# B&R Automation Studio project MotionTestBenchMaster (part 46)

#### Itc_Filler.st
```iecst
ACTION FillerInput:
	(* Commands *)
	VAR_Machine.stFillerModule.iq_stCmd.i_xFillerAbsolutePositionSensor		:= MC_InputOutput.Network.Filler.Commands.FillerAbsolutePositionSensor; (*//V4.A.A.1.6.12e*)
	VAR_Machine.stFillerModule.iq_stCmd.i_xRinserFillerAbsolutePosSensor	:= MC_InputOutput.Network.Filler.Commands.RinserAbsolutePositionSensor; (*//V4.A.A.1.6.12e*)
	VAR_Machine.stFillerModule.iq_stCmd.i_xCapperAbsolutePositionSensor		:= MC_InputOutput.Network.Filler.Commands.CapperAbsolutePositionSensor; (*//V4.A.A.1.6.12e*)
	VAR_Machine.stFillerModule.iq_stCmd.i_xCrownerAbsolutePositionSensor	:= MC_InputOutput.Network.Filler.Commands.CrownerAbsolutePositionSensor; (*//V4.A.A.1.6.12e*)
	VAR_Machine.stFillerModule.iq_stCmd.i_xDoserAbsolutePositionSensor		:= MC_InputOutput.Network.Filler.Commands.DoserAbsolutePositionSensor; (*//V4.A.A.1.6.12e*)

	VAR_Machine.stFillerModule.iq_stCmd.i_xVelocityAxisStop				:= MC_InputOutput.Network.Filler.Commands.VelocityAxisStop;

	FOR uiAxisIndex := CST_FirstFillerModuleAxis TO CST_LastFillerModuleAxis DO
		VAR_Machine.stFillerModule.iq_astSubModuleAxis[uiAxisIndex].iq_stStatus.q_stMainAxisStatus.iq_xNotErrEncoder	:= MC_InputOutput.Safety.Filler.Commands.AxesDiag[uiAxisIndex].DI_NotErrENC;
		VAR_Machine.stFillerModule.iq_astSubModuleAxis[uiAxisIndex].iq_stStatus.q_stMainAxisStatus.iq_xOperational		:= MC_InputOutput.Safety.Filler.Commands.AxesDiag[uiAxisIndex].DI_Operational;
		(* Parameters *)
		IF uiAxisIndex >= 15 THEN
			VAR_Machine.stFillerModule.iq_astSubModuleAxis[uiAxisIndex].iq_stParam.i_rVelocityOffsetFactor		:= MC_InputOutput.Network.Filler.Parameters.OutletConveyorKs / 100.0;
		ELSE
			VAR_Machine.stFillerModule.iq_astSubModuleAxis[uiAxisIndex].iq_stParam.i_rVelocityOffsetFactor		:= MC_InputOutput.Network.Filler.Parameters.InletConveyorKs / 100.0;
		END_IF
	END_FOR

	VAR_Machine.stFillerModule.iq_stParameters.i_uiFillerAbsolutePositionOffset	:= MC_InputOutput.Network.Filler.Parameters.FillerAbsolutePositionOffset; (*//V4.A.A.1.6.12e*)
	VAR_Machine.stFillerModule.iq_stParameters.i_uiFillerStepsNumber			:= MC_InputOutput.Network.Filler.Parameters.FillerStepsNumber; (*//V4.A.A.1.6.12e*)
	VAR_Machine.stFillerModule.iq_stParameters.i_uiRinserAbsolutePositionOffset	:= MC_InputOutput.Network.Filler.Parameters.RinserAbsolutePositionOffset; (*//V4.A.A.1.6.12e*)
	VAR_Machine.stFillerModule.iq_stParameters.i_uiRinserStepsNumber			:= MC_InputOutput.Network.Filler.Parameters.RinserStepsNumber; (*//V4.A.A.1.6.12e*)
	VAR_Machine.stFillerModule.iq_stParameters.i_uiCapperAbsolutePositionOffset	:= MC_InputOutput.Network.Filler.Parameters.CapperAbsolutePositionOffset; (*//V4.A.A.1.6.12e*)
	VAR_Machine.stFillerModule.iq_stParameters.i_uiCapperStepsNumber			:= MC_InputOutput.Network.Filler.Parameters.CapperStepsNumber; (*//V4.A.A.1.6.12e*)
	VAR_Machine.stFillerModule.iq_stParameters.i_uiCrownerAbsolutePosOffset		:= MC_InputOutput.Network.Filler.Parameters.CrownerAbsolutePositionOffset; (*//V4.A.A.1.6.12e*)
	VAR_Machine.stFillerModule.iq_stParameters.i_uiCrownerStepsNumber			:= MC_InputOutput.Network.Filler.Parameters.CrownerStepsNumber; (*//V4.A.A.1.6.12e*)
	VAR_Machine.stFillerModule.iq_stParameters.i_uiDoserPositionOffset			:= MC_InputOutput.Network.Filler.Parameters.DoserAbsolutePositionOffset; (*//V4.A.A.1.6.12e*)
	VAR_Machine.stFillerModule.iq_stParameters.i_uiDoserStepsNumber				:= MC_InputOutput.Network.Filler.Parameters.DoserStepsNumber; (*//V4.A.A.1.6.12e*)

		(*Disable axis Rinser command*)
	VAR_Machine.stFillerModule.iq_astSubModuleAxis[CFG_MC.Mechanical.ReferenceId.Rinser].iq_stCmd.i_xDisableAxis	:= MC_InputOutput.Network.Filler.Commands.DisableRinserAxis;//V4.A.A.1.7.0
	(*Disable axis Doser command*)
	VAR_Machine.stFillerModule.iq_astSubModuleAxis[CFG_MC.Mechanical.ReferenceId.Doser].iq_stCmd.i_xDisableAxis		:= MC_InputOutput.Network.Filler.Commands.DisableDoserAxis;//v999 test
	(*Disable axis Filler command*)
	VAR_Machine.stFillerModule.iq_astSubModuleAxis[CFG_MC.Mechanical.ReferenceId.Filler].iq_stCmd.i_xDisableAxis		:= MC_InputOutput.Network.Filler.Commands.DisableFillerAxis;//v999 test

//	VAR_Machine.stFillerModule.iq_astSubModuleAxis[CST_Inlet10].iq_stCmd.i_xDisableAxis := MC_InputOutput.Network.Filler.Commands.MotorDisableIndex[CST_Inlet10] AND VAR_Machine.stFillerModule.iq_astSubModuleAxis[CST_Inlet10].iq_stStatus.q_stMainAxisStatus.q_xAxisReal;
//	VAR_Machine.stFillerModule.iq_astSubModuleAxis[CST_Inlet09].iq_stCmd.i_xDisableAxis := MC_InputOutput.Network.Filler.Commands.MotorDisableIndex[CST_Inlet09] AND VAR_Machine.stFillerModule.iq_astSubModuleAxis[CST_Inlet09].iq_stStatus.q_stMainAxisStatus.q_xAxisReal;
//	VAR_Machine.stFillerModule.iq_astSubModuleAxis[CST_Inlet08].iq_stCmd.i_xDisableAxis := MC_InputOutput.Network.Filler.Commands.MotorDisableIndex[CST_Inlet08] AND VAR_Machine.stFillerModule.iq_astSubModuleAxis[CST_Inlet08].iq_stStatus.q_stMainAxisStatus.q_xAxisReal;
//	VAR_Machine.stFillerModule.iq_astSubModuleAxis[CST_Inlet07].iq_stCmd.i_xDisableAxis := MC_InputOutput.Network.Filler.Commands.MotorDisableIndex[CST_Inlet07] AND VAR_Machine.stFillerModule.iq_astSubModuleAxis[CST_Inlet07].iq_stStatus.q_stMainAxisStatus.q_xAxisReal;
//	VAR_Machine.stFillerModule.iq_astSubModuleAxis[CST_Inlet06].iq_stCmd.i_xDisableAxis := MC_InputOutput.Network.Filler.Commands.MotorDisableIndex[CST_Inlet06] AND VAR_Machine.stFillerModule.iq_astSubModuleAxis[CST_Inlet06].iq_stStatus.q_stMainAxisStatus.q_xAxisReal;
//	VAR_Machine.stFillerModule.iq_astSubModuleAxis[CST_Inlet05].iq_stCmd.i_xDisableAxis := MC_InputOutput.Network.Filler.Commands.MotorDisableIndex[CST_Inlet05] AND VAR_Machine.stFillerModule.iq_astSubModuleAxis[CST_Inlet05].iq_stStatus.q_stMainAxisStatus.q_xAxisReal;
//	VAR_Machine.stFillerModule.iq_astSubModuleAxis[CST_Inlet04].iq_stCmd.i_xDisableAxis := MC_InputOutput.Network.Filler.Commands.MotorDisableIndex[CST_Inlet04] AND VAR_Machine.stFillerModule.iq_astSubModuleAxis[CST_Inlet04].iq_stStatus.q_stMainAxisStatus.q_xAxisReal;
//	VAR_Machine.stFillerModule.iq_astSubModuleAxis[CST_Inlet03].iq_stCmd.i_xDisableAxis := MC_InputOutput.Network.Filler.Commands.MotorDisableIndex[CST_Inlet03] AND VAR_Machine.stFillerModule.iq_astSubModuleAxis[CST_Inlet03].iq_stStatus.q_stMainAxisStatus.q_xAxisReal;
//	VAR_Machine.stFillerModule.iq_astSubModuleAxis[CST_Inlet02].iq_stCmd.i_xDisableAxis := MC_InputOutput.Network.Filler.Commands.MotorDisableIndex[CST_Inlet02] AND VAR_Machine.stFillerModule.iq_astSubModuleAxis[CST_Inlet02].iq_stStatus.q_stMainAxisStatus.q_xAxisReal;
//	VAR_Machine.stFillerModule.iq_astSubModuleAxis[CST_Inlet01].iq_stCmd.i_xDisableAxis := MC_InputOutput.Network.Filler.Commands.MotorDisableIndex[CST_Inlet01] AND VAR_Machine.stFillerModule.iq_astSubModuleAxis[CST_Inlet01].iq_stStatus.q_stMainAxisStatus.q_xAxisReal;
//	VAR_Machine.stFillerModule.iq_astSubModuleAxis[CST_MainAxis].iq_stCmd.i_xDisableAxis := MC_InputOutput.Network.Filler.Commands.MotorDisableIndex[CST_MainAxis] AND VAR_Machine.stFillerModule.iq_astSubModuleAxis[CST_MainAxis].iq_stStatus.q_stMainAxisStatus.q_xAxisReal;
//	VAR_Machine.stFillerModule.iq_astSubModuleAxis[CST_Outlet01].iq_stCmd.i_xDisableAxis := MC_InputOutput.Network.Filler.Commands.MotorDisableIndex[CST_Outlet01] AND VAR_Machine.stFillerModule.iq_astSubModuleAxis[CST_Outlet01].iq_stStatus.q_stMainAxisStatus.q_xAxisReal;
//	VAR_Machine.stFillerModule.iq_astSubModuleAxis[CST_Outlet02].iq_stCmd.i_xDisableAxis := MC_InputOutput.Network.Filler.Commands.MotorDisableIndex[CST_Outlet02] AND VAR_Machine.stFillerModule.iq_astSubModuleAxis[CST_Outlet02].iq_stStatus.q_stMainAxisStatus.q_xAxisReal;
//	VAR_Machine.stFillerModule.iq_astSubModuleAxis[CST_Outlet03].iq_stCmd.i_xDisableAxis := MC_InputOutput.Network.Filler.Commands.MotorDisableIndex[CST_Outlet03] AND VAR_Machine.stFillerModule.iq_astSubModuleAxis[CST_Outlet03].iq_stStatus.q_stMainAxisStatus.q_xAxisReal;
//	VAR_Machine.stFillerModule.iq_astSubModuleAxis[CST_Outlet04].iq_stCmd.i_xDisableAxis := MC_InputOutput.Network.Filler.Commands.MotorDisableIndex[CST_Outlet04] AND VAR_Machine.stFillerModule.iq_astSubModuleAxis[CST_Outlet04].iq_stStatus.q_stMainAxisStatus.q_xAxisReal;
//	VAR_Machine.stFillerModule.iq_astSubModuleAxis[CST_Outlet05].iq_stCmd.i_xDisableAxis := MC_InputOutput.Network.Filler.Commands.MotorDisableIndex[CST_Outlet05] AND VAR_Machine.stFillerModule.iq_astSubModuleAxis[CST_Outlet05].iq_stStatus.q_stMainAxisStatus.q_xAxisReal;
//	VAR_Machine.stFillerModule.iq_astSubModuleAxis[CST_Outlet06].iq_stCmd.i_xDisableAxis := MC_InputOutput.Network.Filler.Commands.MotorDisableIndex[CST_Outlet06] AND VAR_Machine.stFillerModule.iq_astSubModuleAxis[CST_Outlet06].iq_stStatus.q_stMainAxisStatus.q_xAxisReal;

	VAR_Machine.stFillerModule.iq_astSubModuleAxis[CST_MainAxis].iq_stParam.i_rTorqueErrorThreshold	:= MC_InputOutput.Network.Filler.Parameters.TorqueError.Main;
	FOR uiAxisIndex := 1 TO 10 DO
		VAR_Machine.stFillerModule.iq_astSubModuleAxis[(uiAxisIndex - 1) +  CST_FirstFillerModuleAxis].iq_stParam.i_rTorqueErrorThreshold	:= MC_InputOutput.Network.Filler.Parameters.TorqueError.In[uiAxisIndex];
	END_FOR

	FOR uiAxisIndex := 1 TO 6 DO
		VAR_Machine.stFillerModule.iq_astSubModuleAxis[(uiAxisIndex) + CST_MainAxis].iq_stParam.i_rTorqueErrorThreshold	:= MC_InputOutput.Network.Filler.Parameters.TorqueError.Out[uiAxisIndex];
	END_FOR
END_ACTION

ACTION FillerOutput:
	(* Filler status *)
	MC_InputOutput.Network.Filler.Status.Velocity						:= VAR_Machine.stFillerModule.iq_stStatus.q_rVelocity * 10.0;
	MC_InputOutput.Network.Filler.Status.FillerAbsolutePosition			:= VAR_Machine.stFillerModule.iq_stStatus.q_lrFillerAbsolutePosition; (*//V4.A.A.1.6.12e*)
	MC_InputOutput.Network.Filler.Status.RinserAbsolutePosition			:= VAR_Machine.stFillerModule.iq_stStatus.q_lrRinserAbsolutePosition; (*//V4.A.A.1.6.12e*)
	MC_InputOutput.Network.Filler.Status.CapperAbsolutePosition			:= VAR_Machine.stFillerModule.iq_stStatus.q_lrCapperAbsolutePosition; (*//V4.A.A.1.6.12e*)
	MC_InputOutput.Network.Filler.Status.CrownerAbsolutePosition		:= VAR_Machine.stFillerModule.iq_stStatus.q_lrCrownerAbsolutePosition; (*//V4.A.A.1.6.12e*)
	MC_InputOutput.Network.Filler.Status.DoserAbsolutePosition			:= VAR_Machine.stFillerModule.iq_stStatus.q_lrDoserAbsolutePosition; (*//V4.A.A.1.6.12e*)

	MC_InputOutput.Network.Filler.Status.ModuleHomed					:= VAR_Machine.stFillerModule.iq_stStatus.q_xModuleHomed;
	MC_InputOutput.Network.Filler.Status.ModuleInPosition;
	MC_InputOutput.Network.Filler.Status.ModulePowered					:= VAR_Machine.stFillerModule.iq_stStatus.q_xModulePowered;
	MC_InputOutput.Network.Filler.Status.ModuleReal						:= VAR_Machine.stFillerModule.iq_stStatus.q_xModuleReal;
	MC_InputOutput.Network.Filler.Status.ModuleRunning					:= SEL(VAR_Machine.iq_stStatus.q_xMultiModalityActive, VAR_Machine.iq_stStatus.q_xMachineStartFbk, VAR_Machine.stFillerModule.iq_stStatus.q_xModuleStartFbk);
	MC_InputOutput.Network.Filler.Status.ModuleNotInitialized			:= NOT VAR_Machine.stFillerModule.iq_stStatus.q_xInitDone;

	MC_InputOutput.Network.Filler.Status.AutoActive						:= VAR_Machine.stFillerModule.iq_stStatus.q_xAutoMultiActive;
	MC_InputOutput.Network.Filler.Status.ModuleJogActive				:= VAR_Machine.stFillerModule.iq_stStatus.q_xJogMultiActive;
	MC_InputOutput.Network.Filler.Status.SlowMotionActive				:= VAR_Machine.stFillerModule.iq_stStatus.q_xSlowMotionActive;

	MC_InputOutput.Network.Filler.Status.AutoCmdFeedback				:= VAR_Machine.stFillerModule.iq_stStatus.q_xAutoMultiActive AND VAR_Machine.stFillerModule.iq_stCmd.i_xStart;
	MC_InputOutput.Network.Filler.Status.JogCmdFeedback					:= VAR_Machine.stFillerModule.iq_stStatus.q_xJogMultiActive AND VAR_Machine.stFillerModule.iq_stCmd.i_xJogPB;

	MC_InputOutput.Network.Filler.Status.CarouselReal				:= VAR_Machine.stFillerModule.iq_astSubModuleAxis[CST_MainAxis].iq_stStatus.q_stMainAxisStatus.q_xAxisReal;
	MC_InputOutput.Network.Filler.Status.In01Real					:= VAR_Machine.stFillerModule.iq_astSubModuleAxis[CST_Inlet01].iq_stStatus.q_stMainAxisStatus.q_xAxisReal;
	MC_InputOutput.Network.Filler.Status.In02Real					:= VAR_Machine.stFillerModule.iq_astSubModuleAxis[CST_Inlet02].iq_stStatus.q_stMainAxisStatus.q_xAxisReal;
	MC_InputOutput.Network.Filler.Status.In03Real					:= VAR_Machine.stFillerModule.iq_astSubModuleAxis[CST_Inlet03].iq_stStatus.q_stMainAxisStatus.q_xAxisReal;
	MC_InputOutput.Network.Filler.Status.In04Real					:= VAR_Machine.stFillerModule.iq_astSubModuleAxis[CST_Inlet04].iq_stStatus.q_stMainAxisStatus.q_xAxisReal;
	MC_InputOutput.Network.Filler.Status.In05Real					:= VAR_Machine.stFillerModule.iq_astSubModuleAxis[CST_Inlet05].iq_stStatus.q_stMainAxisStatus.q_xAxisReal;
	MC_InputOutput.Network.Filler.Status.In06Real					:= VAR_Machine.stFillerModule.iq_astSubModuleAxis[CST_Inlet06].iq_stStatus.q_stMainAxisStatus.q_xAxisReal;
	MC_InputOutput.Network.Filler.Status.In07Real					:= VAR_Machine.stFillerModule.iq_astSubModuleAxis[CST_Inlet07].iq_stStatus.q_stMainAxisStatus.q_xAxisReal;
	MC_InputOutput.Network.Filler.Status.In08Real					:= VAR_Machine.stFillerModule.iq_astSubModuleAxis[CST_Inlet08].iq_stStatus.q_stMainAxisStatus.q_xAxisReal;
	MC_InputOutput.Network.Filler.Status.In09Real					:= VAR_Machine.stFillerModule.iq_astSubModuleAxis[CST_Inlet09].iq_stStatus.q_stMainAxisStatus.q_xAxisReal;
	MC_InputOutput.Network.Filler.Status.In10Real					:= VAR_Machine.stFillerModule.iq_astSubModuleAxis[CST_Inlet10].iq_stStatus.q_stMainAxisStatus.q_xAxisReal;
	MC_InputOutput.Network.Filler.Status.Out01Real					:= VAR_Machine.stFillerModule.iq_astSubModuleAxis[CST_Outlet01].iq_stStatus.q_stMainAxisStatus.q_xAxisReal;
	MC_InputOutput.Network.Filler.Status.Out02Real					:= VAR_Machine.stFillerModule.iq_astSubModuleAxis[CST_Outlet02].iq_stStatus.q_stMainAxisStatus.q_xAxisReal;
	MC_InputOutput.Network.Filler.Status.Out03Real					:= VAR_Machine.stFillerModule.iq_astSubModuleAxis[CST_Outlet03].iq_stStatus.q_stMainAxisStatus.q_xAxisReal;
	MC_InputOutput.Network.Filler.Status.Out04Real					:= VAR_Machine.stFillerModule.iq_astSubModuleAxis[CST_Outlet04].iq_stStatus.q_stMainAxisStatus.q_xAxisReal;
	MC_InputOutput.Network.Filler.Status.Out05Real					:= VAR_Machine.stFillerModule.iq_astSubModuleAxis[CST_Outlet05].iq_stStatus.q_stMainAxisStatus.q_xAxisReal;
	MC_InputOutput.Network.Filler.Status.Out06Real					:= VAR_Machine.stFillerModule.iq_astSubModuleAxis[CST_Outlet06].iq_stStatus.q_stMainAxisStatus.q_xAxisReal;

	MC_InputOutput.Network.Filler.Status.FillerAbsolutePositionValid			:= VAR_Machine.stFillerModule.iq_stStatus.q_xFillerAbsolutePositionValid; (*//V4.A.A.1.6.12e*)
	MC_InputOutput.Network.Filler.Status.RinserAbsolutePositionValid			:= VAR_Machine.stFillerModule.iq_stStatus.q_xRinserAbsolutePositionValid; (*//V4.A.A.1.6.12e*)
	MC_InputOutput.Network.Filler.Status.CapperAbsolutePositionValid			:= VAR_Machine.stFillerModule.iq_stStatus.q_xCapperAbsolutePositionValid; (*//V4.A.A.1.6.12e*)
	MC_InputOutput.Network.Filler.Status.CrownerAbsolutePositionValid			:= VAR_Machine.stFillerModule.iq_stStatus.q_xCrownerAbsolutePositionValid; (*//V4.A.A.1.6.12e*)
	MC_InputOutput.Network.Filler.Status.DoserAbsolutePositionValid				:= VAR_Machine.stFillerModule.iq_stStatus.q_xDoserAbsolutePositionValid; (*//V4.A.A.1.6.12e*)

	(* Disable Motor Filler Module Status ----------------------------*)

		(* Disabel Axis FeedBack *) //V4.A.A.1.7.0 Motion
	MC_InputOutput.Network.Filler.Status.DoserAxisDisabled						:= VAR_Machine.stFillerModule.iq_astSubModuleAxis[CFG_MC.Mechanical.ReferenceId.Doser].iq_stStatus.q_stMainAxisStatus.q_xAxisDisabled;
	MC_InputOutput.Network.Filler.Status.RinserAxisDisabled						:= VAR_Machine.stFillerModule.iq_astSubModuleAxis[CFG_MC.Mechanical.ReferenceId.Rinser].iq_stStatus.q_stMainAxisStatus.q_xAxisDisabled;

//	MC_InputOutput.Network.Filler.Status.AxisDisabledFeedBack[CST_Inlet10]		:= VAR_Machine.stFillerModule.iq_astSubModuleAxis[CST_Inlet10].iq_stStatus.q_stMainAxisStatus.q_xAxisDisabled;
//	MC_InputOutput.Network.Filler.Status.AxisDisabledFeedBack[CST_Inlet09]		:= VAR_Machine.stFillerModule.iq_astSubModuleAxis[CST_Inlet09].iq_stStatus.q_stMainAxisStatus.q_xAxisDisabled;
//	MC_InputOutput.Network.Filler.Status.AxisDisabledFeedBack[CST_Inlet08]		:= VAR_Machine.stFillerModule.iq_astSubModuleAxis[CST_Inlet08].iq_stStatus.q_stMainAxisStatus.q_xAxisDisabled;
//	MC_InputOutput.Network.Filler.Status.AxisDisabledFeedBack[CST_Inlet07]		:= VAR_Machine.stFillerModule.iq_astSubModuleAxis[CST_Inlet07].iq_stStatus.q_stMainAxisStatus.q_xAxisDisabled;
//	MC_InputOutput.Network.Filler.Status.AxisDisabledFeedBack[CST_Inlet06]		:= VAR_Machine.stFillerModule.iq_astSubModuleAxis[CST_Inlet06].iq_stStatus.q_stMainAxisStatus.q_xAxisDisabled;
//	MC_InputOutput.Network.Filler.Status.AxisDisabledFeedBack[CST_Inlet05]		:= VAR_Machine.stFillerModule.iq_astSubModuleAxis[CST_Inlet05].iq_stStatus.q_stMainAxisStatus.q_xAxisDisabled;
//	MC_InputOutput.Network.Filler.Status.AxisDisabledFeedBack[CST_Inlet04]		:= VAR_Machine.stFillerModule.iq_astSubModuleAxis[CST_Inlet04].iq_stStatus.q_stMainAxisStatus.q_xAxisDisabled;
//	MC_InputOutput.Network.Filler.Status.AxisDisabledFeedBack[CST_Inlet03]		:= VAR_Machine.stFillerModule.iq_astSubModuleAxis[CST_Inlet03].iq_stStatus.q_stMainAxisStatus.q_xAxisDisabled;
//	MC_InputOutput.Network.Filler.Status.AxisDisabledFeedBack[CST_Inlet02]		:= VAR_Machine.stFillerModule.iq_astSubModuleAxis[CST_Inlet02].iq_stStatus.q_stMainAxisStatus.q_xAxisDisabled;
//	MC_InputOutput.Network.Filler.Status.AxisDisabledFeedBack[CST_Inlet01]		:= VAR_Machine.stFillerModule.iq_astSubModuleAxis[CST_Inlet01].iq_stStatus.q_stMainAxisStatus.q_xAxisDisabled;
//	MC_InputOutput.Network.Filler.Status.AxisDisabledFeedBack[CST_MainAxis]		:= VAR_Machine.stFillerModule.iq_astSubModuleAxis[CST_MainAxis].iq_stStatus.q_stMainAxisStatus.q_xAxisDisabled;
//	MC_InputOutput.Network.Filler.Status.AxisDisabledFeedBack[CST_Outlet01]		:= VAR_Machine.stFillerModule.iq_astSubModuleAxis[CST_Outlet01].iq_stStatus.q_stMainAxisStatus.q_xAxisDisabled;
//	MC_InputOutput.Network.Filler.Status.AxisDisabledFeedBack[CST_Outlet02]		:= VAR_Machine.stFillerModule.iq_astSubModuleAxis[CST_Outlet02].iq_stStatus.q_stMainAxisStatus.q_xAxisDisabled;
//	MC_InputOutput.Network.Filler.Status.AxisDisabledFeedBack[CST_Outlet03]		:= VAR_Machine.stFillerModule.iq_astSubModuleAxis[CST_Outlet03].iq_stStatus.q_stMainAxisStatus.q_xAxisDisabled;
//	MC_InputOutput.Network.Filler.Status.AxisDisabledFeedBack[CST_Outlet04]		:= VAR_Machine.stFillerModule.iq_astSubModuleAxis[CST_Outlet04].iq_stStatus.q_stMainAxisStatus.q_xAxisDisabled;
//	MC_InputOutput.Network.Filler.Status.AxisDisabledFeedBack[CST_Outlet05]		:= VAR_Machine.stFillerModule.iq_astSubModuleAxis[CST_Outlet05].iq_stStatus.q_stMainAxisStatus.q_xAxisDisabled;
//	MC_InputOutput.Network.Filler.Status.AxisDisabledFeedBack[CST_Outlet06]		:= VAR_Machine.stFillerModule.iq_astSubModuleAxis[CST_Outlet06].iq_stStatus.q_stMainAxisStatus.q_xAxisDisabled;

	(* Button Enable *)
	MC_InputOutput.Network.Filler.Status.EnableAutoModality				:= NOT VAR_Machine.stFillerModule.iq_stStatus.q_xReactionActive;
	MC_InputOutput.Network.Filler.Status.EnableJogModality				:= VAR_Machine.stFillerModule.iq_stStatus.q_xModuleStopped AND
																			NOT VAR_Machine.stFillerModule.iq_stStatus.q_xReactionActive;

	(* Exception *)
	(* Main axis exception *)
	MC_InputOutput.Network.Filler.Exceptions.CarouselNotInOpException			:= NOT VAR_Machine.stFillerModule.iq_astSubModuleAxis[CST_MainAxis].iq_stStatus.q_stMainAxisStatus.iq_xOperational;
	MC_InputOutput.Network.Filler.Exceptions.CarouselSafetyException			:= NOT MC_InputOutput.Safety.Filler.Commands.AxesDiag[CST_MainAxis].DI_NotErrFUNC;
	MC_InputOutput.Network.Filler.Exceptions.CarouselTorqueException			:= VAR_Machine.stFillerModule.iq_astSubModuleAxis[CST_MainAxis].iq_stStatus.q_stMainAxisStatus.q_xTorqueError;
	MC_InputOutput.Network.Filler.Exceptions.CarouselTrackException				:= VAR_Machine.stFillerModule.iq_astSubModuleAxis[CST_MainAxis].iq_stStatus.q_stMainAxisStatus.q_xLagError;
	MC_InputOutput.Network.Filler.Exceptions.CarouselDriveException				:= VAR_Machine.stFillerModule.iq_astSubModuleAxis[CST_MainAxis].iq_stStatus.q_stMainAxisStatus.q_xError;
	MC_InputOutput.Network.Filler.Exceptions.CarouselHomeException				:= NOT VAR_Machine.stFillerModule.iq_astSubModuleAxis[CST_MainAxis].iq_stStatus.q_stMainAxisStatus.q_xIsHomed AND
																					VAR_Machine.stFillerModule.iq_astSubModuleAxis[CST_MainAxis].iq_stStatus.q_stMainAxisStatus.q_xInitDone;

	(* Inlet axis exception *)
	IF VAR_Machine.stFillerModule.iq_astSubModuleAxis[CST_Inlet01].iq_stStatus.q_stMainAxisStatus.q_xAxisReal THEN
		IF NOT CFG_MC.Axes.Filler.In[1].VelocityControl THEN
			MC_InputOutput.Network.Filler.Exceptions.Inlet01NotInOpException			:= NOT VAR_Machine.stFillerModule.iq_astSubModuleAxis[CST_Inlet01].iq_stStatus.q_stMainAxisStatus.iq_xOperational;
			MC_InputOutput.Network.Filler.Exceptions.Inlet01SafetyException				:= NOT MC_InputOutput.Safety.Filler.Commands.AxesDiag[CST_Inlet01].DI_NotErrFUNC;
		END_IF
		MC_InputOutput.Network.Filler.Exceptions.Inlet01TorqueException				:= VAR_Machine.stFillerModule.iq_astSubModuleAxis[CST_Inlet01].iq_stStatus.q_stMainAxisStatus.q_xTorqueError;
		MC_InputOutput.Network.Filler.Exceptions.Inlet01TrackException				:= VAR_Machine.stFillerModule.iq_astSubModuleAxis[CST_Inlet01].iq_stStatus.q_stMainAxisStatus.q_xLagError;
		MC_InputOutput.Network.Filler.Exceptions.Inlet01DriveException				:= VAR_Machine.stFillerModule.iq_astSubModuleAxis[CST_Inlet01].iq_stStatus.q_stMainAxisStatus.q_xError;
		MC_InputOutput.Network.Filler.Exceptions.Inlet01HomeException				:= NOT VAR_Machine.stFillerModule.iq_astSubModuleAxis[CST_Inlet01].iq_stStatus.q_stMainAxisStatus.q_xIsHomed AND
																						VAR_Machine.stFillerModule.iq_astSubModuleAxis[CST_Inlet01].iq_stStatus.q_stMainAxisStatus.q_xInitDone;
	END_IF

	IF VAR_Machine.stFillerModule.iq_astSubModuleAxis[CST_Inlet02].iq_stStatus.q_stMainAxisStatus.q_xAxisReal THEN
		IF NOT CFG_MC.Axes.Filler.In[2].VelocityControl THEN
			MC_InputOutput.Network.Filler.Exceptions.Inlet02NotInOpException			:= NOT VAR_Machine.stFillerModule.iq_astSubModuleAxis[CST_Inlet02].iq_stStatus.q_stMainAxisStatus.iq_xOperational;
			MC_InputOutput.Network.Filler.Exceptions.Inlet02SafetyException				:= NOT MC_InputOutput.Safety.Filler.Commands.AxesDiag[CST_Inlet02].DI_NotErrFUNC;
		END_IF
		MC_InputOutput.Network.Filler.Exceptions.Inlet02TorqueException				:= VAR_Machine.stFillerModule.iq_astSubModuleAxis[CST_Inlet02].iq_stStatus.q_stMainAxisStatus.q_xTorqueError;
		MC_InputOutput.Network.Filler.Exceptions.Inlet02TrackException				:= VAR_Machine.stFillerModule.iq_astSubModuleAxis[CST_Inlet02].iq_stStatus.q_stMainAxisStatus.q_xLagError;
		MC_InputOutput.Network.Filler.Exceptions.Inlet02DriveException				:= VAR_Machine.stFillerModule.iq_astSubModuleAxis[CST_Inlet02].iq_stStatus.q_stMainAxisStatus.q_xError;
		MC_InputOutput.Network.Filler.Exceptions.Inlet02HomeException				:= NOT VAR_Machine.stFillerModule.iq_astSubModuleAxis[CST_Inlet02].iq_stStatus.q_stMainAxisStatus.q_xIsHomed AND
																						VAR_Machine.stFillerModule.iq_astSubModuleAxis[CST_Inlet02].iq_stStatus.q_stMainAxisStatus.q_xInitDone;
	END_IF

	IF VAR_Machine.stFillerModule.iq_astSubModuleAxis[CST_Inlet03].iq_stStatus.q_stMainAxisStatus.q_xAxisReal THEN
		IF NOT CFG_MC.Axes.Filler.In[3].VelocityControl THEN
			MC_InputOutput.Network.Filler.Exceptions.Inlet03NotInOpException			:= NOT VAR_Machine.stFillerModule.iq_astSubModuleAxis[CST_Inlet03].iq_stStatus.q_stMainAxisStatus.iq_xOperational;
			MC_InputOutput.Network.Filler.Exceptions.Inlet03SafetyException				:= NOT MC_InputOutput.Safety.Filler.Commands.AxesDiag[CST_Inlet03].DI_NotErrFUNC;
		END_IF
		MC_InputOutput.Network.Filler.Exceptions.Inlet03TorqueException				:= VAR_Machine.stFillerModule.iq_astSubModuleAxis[CST_Inlet03].iq_stStatus.q_stMainAxisStatus.q_xTorqueError;
		MC_InputOutput.Network.Filler.Exceptions.Inlet03TrackException				:= VAR_Machine.stFillerModule.iq_astSubModuleAxis[CST_Inlet03].iq_stStatus.q_stMainAxisStatus.q_xLagError;
		MC_InputOutput.Network.Filler.Exceptions.Inlet03DriveException				:= VAR_Machine.stFillerModule.iq_astSubModuleAxis[CST_Inlet03].iq_stStatus.q_stMainAxisStatus.q_xError;
		MC_InputOutput.Network.Filler.Exceptions.Inlet03HomeException				:= NOT VAR_Machine.stFillerModule.iq_astSubModuleAxis[CST_Inlet03].iq_stStatus.q_stMainAxisStatus.q_xIsHomed AND
																						VAR_Machine.stFillerModule.iq_astSubModuleAxis[CST_Inlet03].iq_stStatus.q_stMainAxisStatus.q_xInitDone;
	END_IF

	IF VAR_Machine.stFillerModule.iq_astSubModuleAxis[CST_Inlet04].iq_stStatus.q_stMainAxisStatus.q_xAxisReal THEN
		IF NOT CFG_MC.Axes.Filler.In[4].VelocityControl THEN
			MC_InputOutput.Network.Filler.Exceptions.Inlet04NotInOpException			:= NOT VAR_Machine.stFillerModule.iq_astSubModuleAxis[CST_Inlet04].iq_stStatus.q_stMainAxisStatus.iq_xOperational;
			MC_InputOutput.Network.Filler.Exceptions.Inlet04SafetyException				:= NOT MC_InputOutput.Safety.Filler.Commands.AxesDiag[CST_Inlet04].DI_NotErrFUNC;
		END_IF
		MC_InputOutput.Network.Filler.Exceptions.Inlet04DriveException				:= VAR_Machine.stFillerModule.iq_astSubModuleAxis[CST_Inlet04].iq_stStatus.q_stMainAxisStatus.q_xError;
		MC_InputOutput.Network.Filler.Exceptions.Inlet04TorqueException				:= VAR_Machine.stFillerModule.iq_astSubModuleAxis[CST_Inlet04].iq_stStatus.q_stMainAxisStatus.q_xTorqueError;
		MC_InputOutput.Network.Filler.Exceptions.Inlet04TrackException				:= VAR_Machine.stFillerModule.iq_astSubModuleAxis[CST_Inlet04].iq_stStatus.q_stMainAxisStatus.q_xLagError;
		MC_InputOutput.Network.Filler.Exceptions.Inlet04HomeException 				:= NOT VAR_Machine.stFillerModule.iq_astSubModuleAxis[CST_Inlet04].iq_stStatus.q_stMainAxisStatus.q_xIsHomed AND
																						VAR_Machine.stFillerModule.iq_astSubModuleAxis[CST_Inlet04].iq_stStatus.q_stMainAxisStatus.q_xInitDone;
	END_IF

	IF VAR_Machine.stFillerModule.iq_astSubModuleAxis[CST_Inlet05].iq_stStatus.q_stMainAxisStatus.q_xAxisReal THEN
		IF NOT CFG_MC.Axes.Filler.In[5].VelocityControl THEN
			MC_InputOutput.Network.Filler.Exceptions.Inlet05NotInOpException			:= NOT VAR_Machine.stFillerModule.iq_astSubModuleAxis[CST_Inlet05].iq_stStatus.q_stMainAxisStatus.iq_xOperational;
			MC_InputOutput.Network.Filler.Exceptions.Inlet05SafetyException				:= NOT MC_InputOutput.Safety.Filler.Commands.AxesDiag[CST_Inlet05].DI_NotErrFUNC;
		END_IF
	MC_InputOutput.Network.Filler.Exceptions.Inlet05DriveException				:= VAR_Machine.stFillerModule.iq_astSubModuleAxis[CST_Inlet05].iq_stStatus.q_stMainAxisStatus.q_xError;
	MC_InputOutput.Network.Filler.Exceptions.Inlet05TorqueException				:= VAR_Machine.stFillerModule.iq_astSubModuleAxis[CST_Inlet05].iq_stStatus.q_stMainAxisStatus.q_xTorqueError;
	MC_InputOutput.Network.Filler.Exceptions.Inlet05TrackException				:= VAR_Machine.stFillerModule.iq_astSubModuleAxis[CST_Inlet05].iq_stStatus.q_stMainAxisStatus.q_xLagError;
	MC_InputOutput.Network.Filler.Exceptions.Inlet05HomeException				:= NOT VAR_Machine.stFillerModule.iq_astSubModuleAxis[CST_Inlet05].iq_stStatus.q_stMainAxisStatus.q_xIsHomed AND
																					VAR_Machine.stFillerModule.iq_astSubModuleAxis[CST_Inlet05].iq_stStatus.q_stMainAxisStatus.q_xInitDone;
	END_IF

	IF VAR_Machine.stFillerModule.iq_astSubModuleAxis[CST_Inlet06].iq_stStatus.q_stMainAxisStatus.q_xAxisReal THEN
		IF NOT CFG_MC.Axes.Filler.In[6].VelocityControl THEN
			MC_InputOutput.Network.Filler.Exceptions.Inlet06NotInOpException			:= NOT VAR_Machine.stFillerModule.iq_astSubModuleAxis[CST_Inlet06].iq_stStatus.q_stMainAxisStatus.iq_xOperational;
			MC_InputOutput.Network.Filler.Exceptions.Inlet06SafetyException				:= NOT MC_InputOutput.Safety.Filler.Commands.AxesDiag[CST_Inlet06].DI_NotErrFUNC;
		END_IF
		MC_InputOutput.Network.Filler.Exceptions.Inlet06DriveException				:= VAR_Machine.stFillerModule.iq_astSubModuleAxis[CST_Inlet06].iq_stStatus.q_stMainAxisStatus.q_xError;
		MC_InputOutput.Network.Filler.Exceptions.Inlet06TorqueException				:= VAR_Machine.stFillerModule.iq_astSubModuleAxis[CST_Inlet06].iq_stStatus.q_stMainAxisStatus.q_xTorqueError;
		MC_InputOutput.Network.Filler.Exceptions.Inlet06TrackException				:= VAR_Machine.stFillerModule.iq_astSubModuleAxis[CST_Inlet06].iq_stStatus.q_stMainAxisStatus.q_xLagError;
		MC_InputOutput.Network.Filler.Exceptions.Inlet06HomeException				:= NOT VAR_Machine.stFillerModule.iq_astSubModuleAxis[CST_Inlet06].iq_stStatus.q_stMainAxisStatus.q_xIsHomed AND
																						VAR_Machine.stFillerModule.iq_astSubModuleAxis[CST_Inlet06].iq_stStatus.q_stMainAxisStatus.q_xInitDone;
	END_IF

	IF VAR_Machine.stFillerModule.iq_astSubModuleAxis[CST_Inlet07].iq_stStatus.q_stMainAxisStatus.q_xAxisReal THEN
		IF NOT CFG_MC.Axes.Filler.In[7].VelocityControl THEN
			MC_InputOutput.Network.Filler.Exceptions.Inlet07NotInOpException			:= NOT VAR_Machine.stFillerModule.iq_astSubModuleAxis[CST_Inlet07].iq_stStatus.q_stMainAxisStatus.iq_xOperational;
			MC_InputOutput.Network.Filler.Exceptions.Inlet07SafetyException				:= NOT MC_InputOutput.Safety.Filler.Commands.AxesDiag[CST_Inlet07].DI_NotErrFUNC;
		END_IF
		MC_InputOutput.Network.Filler.Exceptions.Inlet07DriveException				:= VAR_Machine.stFillerModule.iq_astSubModuleAxis[CST_Inlet07].iq_stStatus.q_stMainAxisStatus.q_xError;
		MC_InputOutput.Network.Filler.Exceptions.Inlet07TorqueException				:= VAR_Machine.stFillerModule.iq_astSubModuleAxis[CST_Inlet07].iq_stStatus.q_stMainAxisStatus.q_xTorqueError;
		MC_InputOutput.Network.Filler.Exceptions.Inlet07TrackException				:= VAR_Machine.stFillerModule.iq_astSubModuleAxis[CST_Inlet07].iq_stStatus.q_stMainAxisStatus.q_xLagError;
		MC_InputOutput.Network.Filler.Exceptions.Inlet07HomeException				:= NOT VAR_Machine.stFillerModule.iq_astSubModuleAxis[CST_Inlet07].iq_stStatus.q_stMainAxisStatus.q_xIsHomed AND
																						VAR_Machine.stFillerModule.iq_astSubModuleAxis[CST_Inlet07].iq_stStatus.q_stMainAxisStatus.q_xInitDone;
	END_IF

	IF VAR_Machine.stFillerModule.iq_astSubModuleAxis[CST_Inlet08].iq_stStatus.q_stMainAxisStatus.q_xAxisReal THEN
		IF NOT CFG_MC.Axes.Filler.In[8].VelocityControl THEN
			MC_InputOutput.Network.Filler.Exceptions.Inlet08NotInOpException			:= NOT VAR_Machine.stFillerModule.iq_astSubModuleAxis[CST_Inlet08].iq_stStatus.q_stMainAxisStatus.iq_xOperational;
			MC_InputOutput.Network.Filler.Exceptions.Inlet08SafetyException				:= NOT MC_InputOutput.Safety.Filler.Commands.AxesDiag[CST_Inlet08].DI_NotErrFUNC;
		END_IF
		MC_InputOutput.Network.Filler.Exceptions.Inlet08DriveException				:= VAR_Machine.stFillerModule.iq_astSubModuleAxis[CST_Inlet08].iq_stStatus.q_stMainAxisStatus.q_xError;
		MC_InputOutput.Network.Filler.Exceptions.Inlet08TorqueException				:= VAR_Machine.stFillerModule.iq_astSubModuleAxis[CST_Inlet08].iq_stStatus.q_stMainAxisStatus.q_xTorqueError;
		MC_InputOutput.Network.Filler.Exceptions.Inlet08TrackException				:= VAR_Machine.stFillerModule.iq_astSubModuleAxis[CST_Inlet08].iq_stStatus.q_stMainAxisStatus.q_xLagError;
		MC_InputOutput.Network.Filler.Exceptions.Inlet08HomeException				:= NOT VAR_Machine.stFillerModule.iq_astSubModuleAxis[CST_Inlet08].iq_stStatus.q_stMainAxisStatus.q_xIsHomed AND
																						VAR_Machine.stFillerModule.iq_astSubModuleAxis[CST_Inlet08].iq_stStatus.q_stMainAxisStatus.q_xInitDone;
	END_IF

	IF VAR_Machine.stFillerModule.iq_astSubModuleAxis[CST_Inlet09].iq_stStatus.q_stMainAxisStatus.q_xAxisReal THEN
		IF NOT CFG_MC.Axes.Filler.In[9].VelocityControl THEN
			MC_InputOutput.Network.Filler.Exceptions.Inlet09NotInOpException			:= NOT VAR_Machine.stFillerModule.iq_astSubModuleAxis[CST_Inlet09].iq_stStatus.q_stMainAxisStatus.iq_xOperational;
			MC_InputOutput.Network.Filler.Exceptions.Inlet09SafetyException				:= NOT MC_InputOutput.Safety.Filler.Commands.AxesDiag[CST_Inlet09].DI_NotErrFUNC;
		END_IF
		MC_InputOutput.Network.Filler.Exceptions.Inlet09DriveException				:= VAR_Machine.stFillerModule.iq_astSubModuleAxis[CST_Inlet09].iq_stStatus.q_stMainAxisStatus.q_xError;
		MC_InputOutput.Network.Filler.Exceptions.Inlet09TorqueException				:= VAR_Machine.stFillerModule.iq_astSubModuleAxis[CST_Inlet09].iq_stStatus.q_stMainAxisStatus.q_xTorqueError;
		MC_InputOutput.Network.Filler.Exceptions.Inlet09TrackException				:= VAR_Machine.stFillerModule.iq_astSubModuleAxis[CST_Inlet09].iq_stStatus.q_stMainAxisStatus.q_xLagError;
		MC_InputOutput.Network.Filler.Exceptions.Inlet09HomeException				:= NOT VAR_Machine.stFillerModule.iq_astSubModuleAxis[CST_Inlet09].iq_stStatus.q_stMainAxisStatus.q_xIsHomed AND
																					VAR_Machine.stFillerModule.iq_astSubModuleAxis[CST_Inlet09].iq_stStatus.q_stMainAxisStatus.q_xInitDone;
	END_IF

	IF VAR_Machine.stFillerModule.iq_astSubModuleAxis[CST_Inlet10].iq_stStatus.q_stMainAxisStatus.q_xAxisReal THEN
		IF NOT CFG_MC.Axes.Filler.In[10].VelocityControl THEN
			MC_InputOutput.Network.Filler.Exceptions.Inlet10NotInOpException			:= NOT VAR_Machine.stFillerModule.iq_astSubModuleAxis[CST_Inlet10].iq_stStatus.q_stMainAxisStatus.iq_xOperational;
			MC_InputOutput.Network.Filler.Exceptions.Inlet10SafetyException				:= NOT MC_InputOutput.Safety.Filler.Commands.AxesDiag[CST_Inlet10].DI_NotErrFUNC;
		END_IF
		MC_InputOutput.Network.Filler.Exceptions.Inlet10DriveException				:= VAR_Machine.stFillerModule.iq_astSubModuleAxis[CST_Inlet10].iq_stStatus.q_stMainAxisStatus.q_xError;
		MC_InputOutput.Network.Filler.Exceptions.Inlet10TorqueException				:= VAR_Machine.stFillerModule.iq_astSubModuleAxis[CST_Inlet10].iq_stStatus.q_stMainAxisStatus.q_xTorqueError;
		MC_InputOutput.Network.Filler.Exceptions.Inlet10TrackException				:= VAR_Machine.stFillerModule.iq_astSubModuleAxis[CST_Inlet10].iq_stStatus.q_stMainAxisStatus.q_xLagError;
		MC_InputOutput.Network.Filler.Exceptions.Inlet10HomeException				:= NOT VAR_Machine.stFillerModule.iq_astSubModuleAxis[CST_Inlet10].iq_stStatus.q_stMainAxisStatus.q_xIsHomed AND
																						VAR_Machine.stFillerModule.iq_astSubModuleAxis[CST_Inlet10].iq_stStatus.q_stMainAxisStatus.q_xInitDone;
	END_IF

	(* Outlet axis exception *)
	IF VAR_Machine.stFillerModule.iq_astSubModuleAxis[CST_Outlet01].iq_stStatus.q_stMainAxisStatus.q_xAxisReal THEN
		IF NOT CFG_MC.Axes.Filler.Out[1].VelocityControl THEN
			MC_InputOutput.Network.Filler.Exceptions.Outlet01NotInOpException			:= NOT VAR_Machine.stFillerModule.iq_astSubModuleAxis[CST_Outlet01].iq_stStatus.q_stMainAxisStatus.iq_xOperational;
			MC_InputOutput.Network.Filler.Exceptions.Outlet01SafetyException			:= NOT MC_InputOutput.Safety.Filler.Commands.AxesDiag[CST_Outlet01].DI_NotErrFUNC;
		END_IF
		MC_InputOutput.Network.Filler.Exceptions.Outlet01DriveException				:= VAR_Machine.stFillerModule.iq_astSubModuleAxis[CST_Outlet01].iq_stStatus.q_stMainAxisStatus.q_xError;
		MC_InputOutput.Network.Filler.Exceptions.Outlet01TorqueException			:= VAR_Machine.stFillerModule.iq_astSubModuleAxis[CST_Outlet01].iq_stStatus.q_stMainAxisStatus.q_xTorqueError;
		MC_InputOutput.Network.Filler.Exceptions.Outlet01TrackException				:= VAR_Machine.stFillerModule.iq_astSubModuleAxis[CST_Outlet01].iq_stStatus.q_stMainAxisStatus.q_xLagError;
		MC_InputOutput.Network.Filler.Exceptions.Outlet01HomeException				:= NOT VAR_Machine.stFillerModule.iq_astSubModuleAxis[CST_Outlet01].iq_stStatus.q_stMainAxisStatus.q_xIsHomed AND
																						VAR_Machine.stFillerModule.iq_astSubModuleAxis[CST_Outlet01].iq_stStatus.q_stMainAxisStatus.q_xInitDone;
	END_IF

	IF VAR_Machine.stFillerModule.iq_astSubModuleAxis[CST_Outlet02].iq_stStatus.q_stMainAxisStatus.q_xAxisReal THEN
		IF NOT CFG_MC.Axes.Filler.Out[2].VelocityControl THEN
			MC_InputOutput.Network.Filler.Exceptions.Outlet02NotInOpException			:= NOT VAR_Machine.stFillerModule.iq_astSubModuleAxis[CST_Outlet02].iq_stStatus.q_stMainAxisStatus.iq_xOperational;
			MC_InputOutput.Network.Filler.Exceptions.Outlet02SafetyException			:= NOT MC_InputOutput.Safety.Filler.Commands.AxesDiag[CST_Outlet02].DI_NotErrFUNC;
		END_IF
		MC_InputOutput.Network.Filler.Exceptions.Outlet02DriveException 			:= VAR_Machine.stFillerModule.iq_astSubModuleAxis[CST_Outlet02].iq_stStatus.q_stMainAxisStatus.q_xError;
		MC_InputOutput.Network.Filler.Exceptions.Outlet02TorqueException			:= VAR_Machine.stFillerModule.iq_astSubModuleAxis[CST_Outlet02].iq_stStatus.q_stMainAxisStatus.q_xTorqueError;
		MC_InputOutput.Network.Filler.Exceptions.Outlet02TrackException 			:= VAR_Machine.stFillerModule.iq_astSubModuleAxis[CST_Outlet02].iq_stStatus.q_stMainAxisStatus.q_xLagError;
		MC_InputOutput.Network.Filler.Exceptions.Outlet02HomeException				:= NOT VAR_Machine.stFillerModule.iq_astSubModuleAxis[CST_Outlet02].iq_stStatus.q_stMainAxisStatus.q_xIsHomed AND
																						VAR_Machine.stFillerModule.iq_astSubModuleAxis[CST_Outlet02].iq_stStatus.q_stMainAxisStatus.q_xInitDone;
	END_IF

	IF VAR_Machine.stFillerModule.iq_astSubModuleAxis[CST_Outlet03].iq_stStatus.q_stMainAxisStatus.q_xAxisReal THEN
		IF NOT CFG_MC.Axes.Filler.Out[3].VelocityControl THEN
			MC_InputOutput.Network.Filler.Exceptions.Outlet03NotInOpException			:= NOT VAR_Machine.stFillerModule.iq_astSubModuleAxis[CST_Outlet03].iq_stStatus.q_stMainAxisStatus.iq_xOperational;
			MC_InputOutput.Network.Filler.Exceptions.Outlet03SafetyException			:= NOT MC_InputOutput.Safety.Filler.Commands.AxesDiag[CST_Outlet03].DI_NotErrFUNC;
		END_IF
		MC_InputOutput.Network.Filler.Exceptions.Outlet03DriveException				:= VAR_Machine.stFillerModule.iq_astSubModuleAxis[CST_Outlet03].iq_stStatus.q_stMainAxisStatus.q_xError;
		MC_InputOutput.Network.Filler.Exceptions.Outlet03TorqueException			:= VAR_Machine.stFillerModule.iq_astSubModuleAxis[CST_Outlet03].iq_stStatus.q_stMainAxisStatus.q_xTorqueError;
		MC_InputOutput.Network.Filler.Exceptions.Outlet03TrackException				:= VAR_Machine.stFillerModule.iq_astSubModuleAxis[CST_Outlet03].iq_stStatus.q_stMainAxisStatus.q_xLagError;
		MC_InputOutput.Network.Filler.Exceptions.Outlet03HomeException				:= NOT VAR_Machine.stFillerModule.iq_astSubModuleAxis[CST_Outlet03].iq_stStatus.q_stMainAxisStatus.q_xIsHomed AND
																						VAR_Machine.stFillerModule.iq_astSubModuleAxis[CST_Outlet03].iq_stStatus.q_stMainAxisStatus.q_xInitDone;
	END_IF

	IF VAR_Machine.stFillerModule.iq_astSubModuleAxis[CST_Outlet04].iq_stStatus.q_stMainAxisStatus.q_xAxisReal THEN
		IF NOT CFG_MC.Axes.Filler.Out[4].VelocityControl THEN
			MC_InputOutput.Network.Filler.Exceptions.Outlet04NotInOpException			:= NOT VAR_Machine.stFillerModule.iq_astSubModuleAxis[CST_Outlet04].iq_stStatus.q_stMainAxisStatus.iq_xOperational;
			MC_InputOutput.Network.Filler.Exceptions.Outlet04SafetyException			:= NOT MC_InputOutput.Safety.Filler.Commands.AxesDiag[CST_Outlet04].DI_NotErrFUNC;
		END_IF
		MC_InputOutput.Network.Filler.Exceptions.Outlet04DriveException 			:= VAR_Machine.stFillerModule.iq_astSubModuleAxis[CST_Outlet04].iq_stStatus.q_stMainAxisStatus.q_xError;
		MC_InputOutput.Network.Filler.Exceptions.Outlet04TorqueException			:= VAR_Machine.stFillerModule.iq_astSubModuleAxis[CST_Outlet04].iq_stStatus.q_stMainAxisStatus.q_xTorqueError;
		MC_InputOutput.Network.Filler.Exceptions.Outlet04TrackException 			:= VAR_Machine.stFillerModule.iq_astSubModuleAxis[CST_Outlet04].iq_stStatus.q_stMainAxisStatus.q_xLagError;
		MC_InputOutput.Network.Filler.Exceptions.Outlet04HomeException				:= NOT VAR_Machine.stFillerModule.iq_astSubModuleAxis[CST_Outlet04].iq_stStatus.q_stMainAxisStatus.q_xIsHomed AND
																						VAR_Machine.stFillerModule.iq_astSubModuleAxis[CST_Outlet04].iq_stStatus.q_stMainAxisStatus.q_xInitDone;
	END_IF

	IF VAR_Machine.stFillerModule.iq_astSubModuleAxis[CST_Outlet05].iq_stStatus.q_stMainAxisStatus.q_xAxisReal THEN
		IF NOT CFG_MC.Axes.Filler.Out[5].VelocityControl THEN
			MC_InputOutput.Network.Filler.Exceptions.Outlet05NotInOpException			:= NOT VAR_Machine.stFillerModule.iq_astSubModuleAxis[CST_Outlet05].iq_stStatus.q_stMainAxisStatus.iq_xOperational;
			MC_InputOutput.Network.Filler.Exceptions.Outlet05SafetyException			:= NOT MC_InputOutput.Safety.Filler.Commands.AxesDiag[CST_Outlet05].DI_NotErrFUNC;
		END_IF
		MC_InputOutput.Network.Filler.Exceptions.Outlet05DriveException				:= VAR_Machine.stFillerModule.iq_astSubModuleAxis[CST_Outlet05].iq_stStatus.q_stMainAxisStatus.q_xError;
		MC_InputOutput.Network.Filler.Exceptions.Outlet05TorqueException			:= VAR_Machine.stFillerModule.iq_astSubModuleAxis[CST_Outlet05].iq_stStatus.q_stMainAxisStatus.q_xTorqueError;
		MC_InputOutput.Network.Filler.Exceptions.Outlet05TrackException				:= VAR_Machine.stFillerModule.iq_astSubModuleAxis[CST_Outlet05].iq_stStatus.q_stMainAxisStatus.q_xLagError;
		MC_InputOutput.Network.Filler.Exceptions.Outlet05HomeException				:= NOT VAR_Machine.stFillerModule.iq_astSubModuleAxis[CST_Outlet05].iq_stStatus.q_stMainAxisStatus.q_xIsHomed AND
																						VAR_Machine.stFillerModule.iq_astSubModuleAxis[CST_Outlet05].iq_stStatus.q_stMainAxisStatus.q_xInitDone;
	END_IF

	IF VAR_Machine.stFillerModule.iq_astSubModuleAxis[CST_Outlet06].iq_stStatus.q_stMainAxisStatus.q_xAxisReal THEN
		IF NOT CFG_MC.Axes.Filler.Out[6].VelocityControl THEN
			MC_InputOutput.Network.Filler.Exceptions.Outlet06NotInOpException			:= NOT VAR_Machine.stFillerModule.iq_astSubModuleAxis[CST_Outlet06].iq_stStatus.q_stMainAxisStatus.iq_xOperational;
			MC_InputOutput.Network.Filler.Exceptions.Outlet06SafetyException			:= NOT MC_InputOutput.Safety.Filler.Commands.AxesDiag[CST_Outlet06].DI_NotErrFUNC;
		END_IF
		MC_InputOutput.Network.Filler.Exceptions.Outlet06DriveException 			:= VAR_Machine.stFillerModule.iq_astSubModuleAxis[CST_Outlet06].iq_stStatus.q_stMainAxisStatus.q_xError;
		MC_InputOutput.Network.Filler.Exceptions.Outlet06TorqueException			:= VAR_Machine.stFillerModule.iq_astSubModuleAxis[CST_Outlet06].iq_stStatus.q_stMainAxisStatus.q_xTorqueError;
		MC_InputOutput.Network.Filler.Exceptions.Outlet06TrackException 			:= VAR_Machine.stFillerModule.iq_astSubModuleAxis[CST_Outlet06].iq_stStatus.q_stMainAxisStatus.q_xLagError;
		MC_InputOutput.Network.Filler.Exceptions.Outlet06HomeException				:= NOT VAR_Machine.stFillerModule.iq_astSubModuleAxis[CST_Outlet06].iq_stStatus.q_stMainAxisStatus.q_xIsHomed AND
																						VAR_Machine.stFillerModule.iq_astSubModuleAxis[CST_Outlet06].iq_stStatus.q_stMainAxisStatus.q_xInitDone;
	END_IF
END_ACTION
```

#### Itc_Outlet.st
```iecst
ACTION OutletInput:
	(* Commands *)
	VAR_Machine.stOutletModule.iq_stCmd.i_xVelocityAxisStop			:= MC_InputOutput.Network.Outlet.Commands.VelocityAxisStop;

	FOR uiAxisIndex := CST_FirstOutletModuleAxis TO CST_LastOutletModuleAxis DO
		VAR_Machine.stOutletModule.iq_astSubModuleAxis[uiAxisIndex].iq_stStatus.q_stMainAxisStatus.iq_xNotErrEncoder	:= MC_InputOutput.Safety.Outlet.Commands.AxesDiag[uiAxisIndex].DI_NotErrENC;
		VAR_Machine.stOutletModule.iq_astSubModuleAxis[uiAxisIndex].iq_stStatus.q_stMainAxisStatus.iq_xOperational		:= MC_InputOutput.Safety.Outlet.Commands.AxesDiag[uiAxisIndex].DI_Operational;
	(* Parameters *)
		IF uiAxisIndex > 15 THEN
			VAR_Machine.stOutletModule.iq_astSubModuleAxis[uiAxisIndex].iq_stParam.i_rVelocityOffsetFactor	:= MC_InputOutput.Network.Outlet.Parameters.ConveyorKs / 100.0;
		ELSE
			VAR_Machine.stOutletModule.iq_astSubModuleAxis[uiAxisIndex].iq_stParam.i_rVelocityOffsetFactor	:= MC_InputOutput.Network.Outlet.Parameters.ConveyorKs / 100.0;
		END_IF
	END_FOR

END_ACTION

ACTION OutletOutput:
	(* Outlet status *)
	MC_InputOutput.Network.Outlet.Status.Velocity							:= VAR_Machine.stOutletModule.iq_stStatus.q_rVelocity * 10.0;

	MC_InputOutput.Network.Outlet.Status.ModuleHomed						:= VAR_Machine.stOutletModule.iq_stStatus.q_xModuleHomed;
	MC_InputOutput.Network.Outlet.Status.ModuleInPosition;
	MC_InputOutput.Network.Outlet.Status.ModulePowered						:= VAR_Machine.stOutletModule.iq_stStatus.q_xModulePowered;
	MC_InputOutput.Network.Outlet.Status.ModuleReal							:= VAR_Machine.stOutletModule.iq_stStatus.q_xModuleReal;
	MC_InputOutput.Network.Outlet.Status.ModuleRunning						:= SEL(VAR_Machine.iq_stStatus.q_xMultiModalityActive, VAR_Machine.iq_stStatus.q_xMachineStartFbk, VAR_Machine.stOutletModule.iq_stStatus.q_xModuleStartFbk);
	MC_InputOutput.Network.Outlet.Status.ModuleNotInitialized				:= NOT VAR_Machine.stOutletModule.iq_stStatus.q_xInitDone;

	MC_InputOutput.Network.Outlet.Status.AutoActive							:= VAR_Machine.stOutletModule.iq_stStatus.q_xAutoMultiActive;
	MC_InputOutput.Network.Outlet.Status.ModuleJogActive					:= VAR_Machine.stOutletModule.iq_stStatus.q_xJogMultiActive;
	MC_InputOutput.Network.Outlet.Status.SlowMotionActive					:= VAR_Machine.stOutletModule.iq_stStatus.q_xSlowMotionActive;

	MC_InputOutput.Network.Outlet.Status.AutoCmdFeedback					:= VAR_Machine.stOutletModule.iq_stStatus.q_xAutoMultiActive AND VAR_Machine.stOutletModule.iq_stCmd.i_xStart;
	MC_InputOutput.Network.Outlet.Status.JogCmdFeedback						:= VAR_Machine.stOutletModule.iq_stStatus.q_xJogMultiActive AND VAR_Machine.stOutletModule.iq_stCmd.i_xJogPB;

	MC_InputOutput.Network.Outlet.Status.MainAxisReal						:= VAR_Machine.stOutletModule.iq_astSubModuleAxis[CST_MainAxis].iq_stStatus.q_stMainAxisStatus.q_xAxisReal;
	MC_InputOutput.Network.Outlet.Status.Out01Real							:= VAR_Machine.stOutletModule.iq_astSubModuleAxis[CST_Outlet01].iq_stStatus.q_stMainAxisStatus.q_xAxisReal;
	MC_InputOutput.Network.Outlet.Status.Out02Real							:= VAR_Machine.stOutletModule.iq_astSubModuleAxis[CST_Outlet02].iq_stStatus.q_stMainAxisStatus.q_xAxisReal;
	MC_InputOutput.Network.Outlet.Status.Out03Real							:= VAR_Machine.stOutletModule.iq_astSubModuleAxis[CST_Outlet03].iq_stStatus.q_stMainAxisStatus.q_xAxisReal;
	MC_InputOutput.Network.Outlet.Status.Out04Real							:= VAR_Machine.stOutletModule.iq_astSubModuleAxis[CST_Outlet04].iq_stStatus.q_stMainAxisStatus.q_xAxisReal;

	(* Button Enable *)
	MC_InputOutput.Network.Outlet.Status.EnableAutoModality					:= NOT VAR_Machine.stOutletModule.iq_stStatus.q_xReactionActive;
	MC_InputOutput.Network.Outlet.Status.EnableJogModality					:= VAR_Machine.stOutletModule.iq_stStatus.q_xModuleStopped AND
																				NOT VAR_Machine.stOutletModule.iq_stStatus.q_xReactionActive;

	(* Exception *)
	(* Main axis exception *)
	IF VAR_Machine.stOutletModule.iq_astSubModuleAxis[CST_MainAxis].iq_stStatus.q_stMainAxisStatus.q_xAxisReal THEN
		MC_InputOutput.Network.Outlet.Exceptions.MainAxisNotInOpException		:= NOT VAR_Machine.stOutletModule.iq_astSubModuleAxis[CST_MainAxis].iq_stStatus.q_stMainAxisStatus.iq_xOperational;
		MC_InputOutput.Network.Outlet.Exceptions.MainAxisSafetyException		:= NOT MC_InputOutput.Safety.Outlet.Commands.AxesDiag[CST_MainAxis].DI_NotErrFUNC;
		MC_InputOutput.Network.Outlet.Exceptions.MainAxisDriveException			:= VAR_Machine.stOutletModule.iq_astSubModuleAxis[CST_MainAxis].iq_stStatus.q_stMainAxisStatus.q_xError;
		MC_InputOutput.Network.Outlet.Exceptions.MainAxisTorqueException		:= VAR_Machine.stOutletModule.iq_astSubModuleAxis[CST_MainAxis].iq_stStatus.q_stMainAxisStatus.q_xTorqueError;
		MC_InputOutput.Network.Outlet.Exceptions.MainAxisTrackException			:= VAR_Machine.stOutletModule.iq_astSubModuleAxis[CST_MainAxis].iq_stStatus.q_stMainAxisStatus.q_xLagError;
		MC_InputOutput.Network.Outlet.Exceptions.MainAxisHomeException			:= NOT VAR_Machine.stOutletModule.iq_astSubModuleAxis[CST_MainAxis].iq_stStatus.q_stMainAxisStatus.q_xIsHomed AND
																				VAR_Machine.stOutletModule.iq_astSubModuleAxis[CST_MainAxis].iq_stStatus.q_stMainAxisStatus.q_xInitDone;
	END_IF

	(* Outlet axis exception *)
	IF VAR_Machine.stOutletModule.iq_astSubModuleAxis[CST_Outlet01].iq_stStatus.q_stMainAxisStatus.q_xAxisReal THEN
		IF NOT CFG_MC.Axes.Outlet.Out[1].VelocityControl THEN
			MC_InputOutput.Network.Outlet.Exceptions.Outlet01NotInOpException		:= NOT VAR_Machine.stOutletModule.iq_astSubModuleAxis[CST_Outlet01].iq_stStatus.q_stMainAxisStatus.iq_xOperational;
			MC_InputOutput.Network.Outlet.Exceptions.Outlet01SafetyException		:= NOT MC_InputOutput.Safety.Outlet.Commands.AxesDiag[CST_Outlet01].DI_NotErrFUNC;
		END_IF
		MC_InputOutput.Network.Outlet.Exceptions.Outlet01DriveException				:= VAR_Machine.stOutletModule.iq_astSubModuleAxis[CST_Outlet01].iq_stStatus.q_stMainAxisStatus.q_xError;
		MC_InputOutput.Network.Outlet.Exceptions.Outlet01TorqueException			:= VAR_Machine.stOutletModule.iq_astSubModuleAxis[CST_Outlet01].iq_stStatus.q_stMainAxisStatus.q_xTorqueError;
		MC_InputOutput.Network.Outlet.Exceptions.Outlet01TrackException				:= VAR_Machine.stOutletModule.iq_astSubModuleAxis[CST_Outlet01].iq_stStatus.q_stMainAxisStatus.q_xLagError;
		MC_InputOutput.Network.Outlet.Exceptions.Outlet01HomeException				:= NOT VAR_Machine.stOutletModule.iq_astSubModuleAxis[CST_Outlet01].iq_stStatus.q_stMainAxisStatus.q_xIsHomed AND
																						VAR_Machine.stOutletModule.iq_astSubModuleAxis[CST_Outlet01].iq_stStatus.q_stMainAxisStatus.q_xInitDone;
	END_IF

	IF VAR_Machine.stOutletModule.iq_astSubModuleAxis[CST_Outlet02].iq_stStatus.q_stMainAxisStatus.q_xAxisReal THEN
		IF NOT CFG_MC.Axes.Outlet.Out[2].VelocityControl THEN
			MC_InputOutput.Network.Outlet.Exceptions.Outlet02NotInOpException		:= NOT VAR_Machine.stOutletModule.iq_astSubModuleAxis[CST_Outlet02].iq_stStatus.q_stMainAxisStatus.iq_xOperational;
			MC_InputOutput.Network.Outlet.Exceptions.Outlet02SafetyException		:= NOT MC_InputOutput.Safety.Outlet.Commands.AxesDiag[CST_Outlet02].DI_NotErrFUNC;
		END_IF
		MC_InputOutput.Network.Outlet.Exceptions.Outlet02DriveException 			:= VAR_Machine.stOutletModule.iq_astSubModuleAxis[CST_Outlet02].iq_stStatus.q_stMainAxisStatus.q_xError;
		MC_InputOutput.Network.Outlet.Exceptions.Outlet02TorqueException			:= VAR_Machine.stOutletModule.iq_astSubModuleAxis[CST_Outlet02].iq_stStatus.q_stMainAxisStatus.q_xTorqueError;
		MC_InputOutput.Network.Outlet.Exceptions.Outlet02TrackException 			:= VAR_Machine.stOutletModule.iq_astSubModuleAxis[CST_Outlet02].iq_stStatus.q_stMainAxisStatus.q_xLagError;
		MC_InputOutput.Network.Outlet.Exceptions.Outlet02HomeException				:= NOT VAR_Machine.stOutletModule.iq_astSubModuleAxis[CST_Outlet02].iq_stStatus.q_stMainAxisStatus.q_xIsHomed AND
																						VAR_Machine.stOutletModule.iq_astSubModuleAxis[CST_Outlet02].iq_stStatus.q_stMainAxisStatus.q_xInitDone;
	END_IF

	IF VAR_Machine.stOutletModule.iq_astSubModuleAxis[CST_Outlet03].iq_stStatus.q_stMainAxisStatus.q_xAxisReal THEN
		IF NOT CFG_MC.Axes.Outlet.Out[3].VelocityControl THEN
			MC_InputOutput.Network.Outlet.Exceptions.Outlet03NotInOpException		:= NOT VAR_Machine.stOutletModule.iq_astSubModuleAxis[CST_Outlet03].iq_stStatus.q_stMainAxisStatus.iq_xOperational;
			MC_InputOutput.Network.Outlet.Exceptions.Outlet03SafetyException		:= NOT MC_InputOutput.Safety.Outlet.Commands.AxesDiag[CST_Outlet03].DI_NotErrFUNC;
		END_IF
		MC_InputOutput.Network.Outlet.Exceptions.Outlet03DriveException				:= VAR_Machine.stOutletModule.iq_astSubModuleAxis[CST_Outlet03].iq_stStatus.q_stMainAxisStatus.q_xError;
		MC_InputOutput.Network.Outlet.Exceptions.Outlet03TorqueException			:= VAR_Machine.stOutletModule.iq_astSubModuleAxis[CST_Outlet03].iq_stStatus.q_stMainAxisStatus.q_xTorqueError;
		MC_InputOutput.Network.Outlet.Exceptions.Outlet03TrackException				:= VAR_Machine.stOutletModule.iq_astSubModuleAxis[CST_Outlet03].iq_stStatus.q_stMainAxisStatus.q_xLagError;
		MC_InputOutput.Network.Outlet.Exceptions.Outlet03HomeException				:= NOT VAR_Machine.stOutletModule.iq_astSubModuleAxis[CST_Outlet03].iq_stStatus.q_stMainAxisStatus.q_xIsHomed AND
																						VAR_Machine.stOutletModule.iq_astSubModuleAxis[CST_Outlet03].iq_stStatus.q_stMainAxisStatus.q_xInitDone;
	END_IF

	IF VAR_Machine.stOutletModule.iq_astSubModuleAxis[CST_Outlet04].iq_stStatus.q_stMainAxisStatus.q_xAxisReal THEN
		IF NOT CFG_MC.Axes.Outlet.Out[4].VelocityControl THEN
			MC_InputOutput.Network.Outlet.Exceptions.Outlet04NotInOpException		:= NOT VAR_Machine.stOutletModule.iq_astSubModuleAxis[CST_Outlet04].iq_stStatus.q_stMainAxisStatus.iq_xOperational;
			MC_InputOutput.Network.Outlet.Exceptions.Outlet04SafetyException		:= NOT MC_InputOutput.Safety.Outlet.Commands.AxesDiag[CST_Outlet04].DI_NotErrFUNC;
		END_IF
		MC_InputOutput.Network.Outlet.Exceptions.Outlet04DriveException 			:= VAR_Machine.stOutletModule.iq_astSubModuleAxis[CST_Outlet04].iq_stStatus.q_stMainAxisStatus.q_xError;
		MC_InputOutput.Network.Outlet.Exceptions.Outlet04TorqueException			:= VAR_Machine.stOutletModule.iq_astSubModuleAxis[CST_Outlet04].iq_stStatus.q_stMainAxisStatus.q_xTorqueError;
		MC_InputOutput.Network.Outlet.Exceptions.Outlet04TrackException 			:= VAR_Machine.stOutletModule.iq_astSubModuleAxis[CST_Outlet04].iq_stStatus.q_stMainAxisStatus.q_xLagError;
		MC_InputOutput.Network.Outlet.Exceptions.Outlet04HomeException				:= NOT VAR_Machine.stOutletModule.iq_astSubModuleAxis[CST_Outlet04].iq_stStatus.q_stMainAxisStatus.q_xIsHomed AND
																						VAR_Machine.stOutletModule.iq_astSubModuleAxis[CST_Outlet04].iq_stStatus.q_stMainAxisStatus.q_xInitDone;
	END_IF
END_ACTION
```

### Program Logical/30_MC/Task/Cyclic05/MC_IDLE (IEC) - MC_IDLE - C#5 20ms

#### Cyclic.st - Cyclic code
```iecst
PROGRAM _CYCLIC
(***** FUBs cyclic call *****)
	fbMpAlarmXListUI_Main();

	(* Hmi management *)
	tonUpdateHmiUi.PT	:= t#10s;
	tonUpdateHmiUi.IN	:= NOT xUpdateUi;
	tonUpdateHmiUi();

	stMainUIConnect.AcknowledgeAll	:= MC_InputOutput.Network.Machine.Commands.AlarmReset;

	IF tonUpdateHmiUi.Q THEN
		xUpdateUi	:= TRUE;
	END_IF

	IF xUpdateUi THEN
		IF strlen(ADR(stMainUIConnect.AlarmList.Message[uiStringCounter]))> 0 THEN
			strcpy(ADR(HMI_MC_AlarmList[uiStringCounter]),ADR(stMainUIConnect.AlarmList.Message[uiStringCounter]));
		ELSIF strlen(ADR(stMainUIConnect.AlarmList.Name[uiStringCounter]))> 0 THEN
			strcpy(ADR(HMI_MC_AlarmList[uiStringCounter]),ADR(stMainUIConnect.AlarmList.Name[uiStringCounter]));
		ELSE
			HMI_MC_AlarmList[uiStringCounter]:= '';
		END_IF

		uiStringCounter := (uiStringCounter + 1) MOD 10;

		IF uiStringCounter = 0 THEN
			xUpdateUi	:= FALSE;
		END_IF
	ELSE
		uiStringCounter	:= 0;
	END_IF
END_PROGRAM
```

#### Init.st - Init code
```iecst
PROGRAM _INIT
	(* AlarmX UI Setup *)
	stMainAlarmSetup.AlarmListScrollWindow	:= 0;
	stMainAlarmSetup.AlarmListSize			:= 100;

	(* AlarmX UI Connect *)
	stMainUIConnect;

	(* Ui Init *)
	fbMpAlarmXListUI_Main.MpLink		:= ADR(gMainAlarmXCoreLink);
	fbMpAlarmXListUI_Main.UISetup		:= stMainAlarmSetup;
	fbMpAlarmXListUI_Main.UIConnect		:= ADR(stMainUIConnect);
	fbMpAlarmXListUI_Main.Enable		:= TRUE;
END_PROGRAM
```

#### Variables.var - Local variables
```iecst
(*Main*)
VAR
	tonUpdateHmiUi : TON;
	xUpdateUi : BOOL;
	uiStringCounter : UINT;
	stMainUIConnect : MpAlarmXListUIConnectType := (0);
	fbMpAlarmXListUI_Main : MpAlarmXListUI;
	stMainAlarmSetup : MpAlarmXListUISetupType;
END_VAR
```

### CFG_Variables.var
```iecst
VAR
	CFG_MC : CFG_Motion_Type;
END_VAR
```

### CFG_Types.typ
```iecst
TYPE
	CFG_Motion_Type : 	STRUCT
		Generic : CFG_Generic_Type;
		Mechanical : CFG_Mechanical_Type;
		MotorDisableConfig : ARRAY[0..9]OF CFG_MotorDisableConfig_Type;
		Movements : CFG_Movements_Type;
		MaximumGearBoxTorque : CFG_Torque_Type;
		Axes : CFG_Axes_Type;
	END_STRUCT;
	CFG_Generic_Type : 	STRUCT
		KochModulePresent : BOOL;
		DisengageImmediately : BOOL; (*In combi mode if TRUE disengage immediately the machine, without waiting SynchroDisengage command*)
		AxesMultiplexingOn : BOOL;
		MotionIntegrated : BOOL;
		SyncroPar : CFG_SyncroPar_Type;
		Aseptic : BOOL;
		DoubleInlet : BOOL; (*If TRUE Inlet03 and Inlet06 take Inlet02 as Homing Master*)
		EmulationCardPulses : UINT;
	END_STRUCT;
	CFG_SyncroPar_Type : 	STRUCT
		ExternalEncoder : BOOL;
		ExternalPositionFormat : BOOL; (*FALSE: LREAL TRUE: DINT //v4.A.A.1.7.0*)
		NumberOfSteps : UINT; (*Master Virtual Position := 1*)
		ExternalSignalPeriod : UDINT; (*Master Virtual Position := 3600000*)
	END_STRUCT;
	CFG_Mechanical_Type : 	STRUCT
		MachineStep : LREAL; (*Machine Step [mm]*)
		LagErrorThreshold : REAL; (*Lag error threshold [mm]*)
		ReferenceId : CFG_RefId_Type;
	END_STRUCT;
	CFG_RefId_Type : 	STRUCT
		Capper : USINT;
		Crowner : USINT;
		Doser : USINT;
		Filler : USINT;
		Rinser : USINT;
		Seamer : USINT;
	END_STRUCT;
	CFG_Movements_Type : 	STRUCT
		Jerk : REAL;
		EmergencyDec : REAL;
		ShutDownDec : REAL;
		MachineMaxSpeed : REAL;
	END_STRUCT;
	CFG_MotorDisableConfig_Type : 	STRUCT
		MotorIndexNumberDisable : ARRAY[CST_FirstFillerModuleAxis..CST_LastFillerModuleAxis]OF BOOL;
	END_STRUCT;
	CFG_Torque_Type : 	STRUCT
		Inlet : CFG_InletTorque_Type;
		Filler : CFG_FillerTorque_Type;
		Outlet : CFG_OutletTorque_Type;
	END_STRUCT;
	CFG_InletTorque_Type : 	STRUCT
		Main : REAL;
		In : ARRAY[1..4]OF REAL;
		Out : ARRAY[1..4]OF REAL;
	END_STRUCT;
	CFG_FillerTorque_Type : 	STRUCT
		Main : REAL;
		In : ARRAY[1..10]OF REAL;
		Out : ARRAY[1..6]OF REAL;
	END_STRUCT;
	CFG_OutletTorque_Type : 	STRUCT
		Main : REAL;
		In : ARRAY[1..4]OF REAL;
		Out : ARRAY[1..4]OF REAL;
	END_STRUCT;
	CFG_Axes_Type : 	STRUCT
		Inlet : CFG_InletAxes_Type;
		Filler : CFG_FillerAxes_Type;
		Outlet : CFG_OutletAxes_Type;
	END_STRUCT;
	CFG_InletAxes_Type : 	STRUCT
		Main : CFG_Axis_Type;
		In : ARRAY[1..4]OF CFG_Axis_Type;
		Out : ARRAY[1..4]OF CFG_Axis_Type;
	END_STRUCT;
	CFG_FillerAxes_Type : 	STRUCT
		Main : CFG_Axis_Type;
		In : ARRAY[1..10]OF CFG_Axis_Type;
		Out : ARRAY[1..6]OF CFG_Axis_Type;
	END_STRUCT;
	CFG_OutletAxes_Type : 	STRUCT
		Main : CFG_Axis_Type;
		In : ARRAY[1..4]OF CFG_Axis_Type;
		Out : ARRAY[1..4]OF CFG_Axis_Type;
	END_STRUCT;
	CFG_Axis_Type : 	STRUCT
		HmiNameId : USINT;
		ThirdPartyMotor : BOOL;
		VelocityControl : BOOL;
		InductionMotor : BOOL;
		InductionMotorData : CFG_InductionMotorSetup_Type;
	END_STRUCT;
	CFG_InductionMotorSetup_Type : 	STRUCT
		RatedVoltage : REAL; (*rated voltage [V]*)
		RatedCurrent : REAL; (*rated current [A]*)
		RatedSpeed : REAL; (*rated numbers of revolutions [1/min]*)
		RatedFrequency : REAL; (*rated frequenzy [Hz]*)
		PowerFactor : REAL; (*cos phi*)
		ThermalTrippingTime : REAL; (*tripping time at thermal overload [s]*)
	END_STRUCT;
END_TYPE
```

### Package Logical/31_DOS - Doser:gestione per aromi e polpe

### Program Logical/31_DOS/DOS (IEC) - DOS Main Program - C#4 - 100ms

#### DOS.sfc - Cyclic code
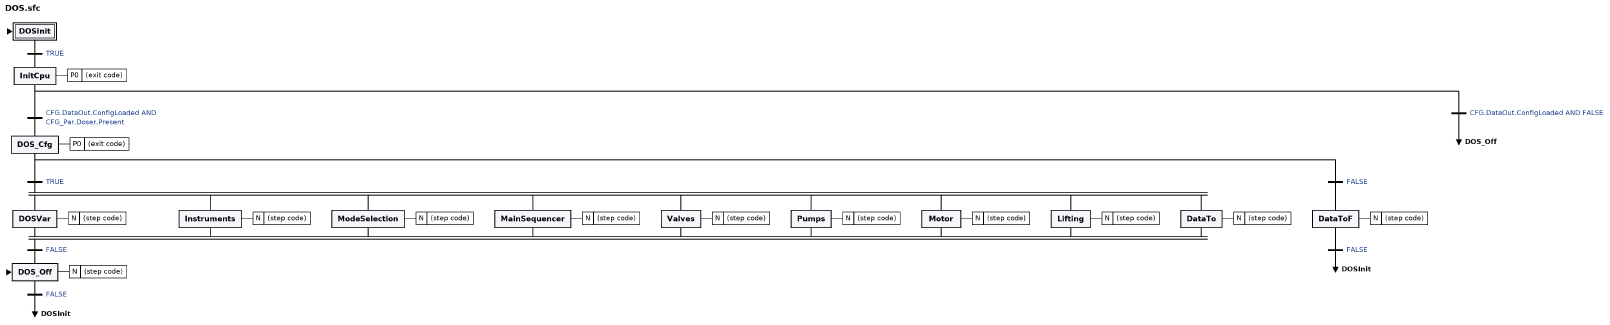
```iecst
PROGRAM _CYCLIC
INITIAL_STEP DOSInit:
END_STEP
TRANSITION FROM DOSInit TO InitCpu:=
TRUE
END_TRANSITION
STEP InitCpu:
END_STEP
EXIT_ACTION

END_ACTION
TRANSITION PRESENT FROM InitCpu TO DOS_Cfg:=
CFG.DataOut.ConfigLoaded AND CFG_Par.Doser.Present //RMH017
END_TRANSITION
TRANSITION NOT PRESENT FROM InitCpu TO DOS_Off:=
CFG.DataOut.ConfigLoaded AND FALSE //V4.A.A.1.6.11 : WAITING FOR CFG
END_TRANSITION
(* @SFCISJUMP := 'DOS_Off' *)
STEP DOS_Cfg:
END_STEP
EXIT_ACTION
DOS_Hardware_CFG;

//Gestione HMI RMH017
HMI_CFG_PAR_1._005 := FALSE; //FLAVOR DOSER
HMI_CFG_PAR_1._215 := TRUE;
HMI_CFG_PAR_1._216 := TRUE; //PULP DOSER
HMI_CFG_PAR_1._217 := MMJ[201].IN_ConfigPresent;
HMI_CFG_PAR_1._218 := MMJ[201].IN_ConfigPresent;

HMI_CFG_PAM_A1._400 := PPJ203.IN_ConfigPresent;
HMI_CFG_PAM_A1._401 := PPJ203.IN_ConfigPresent;
HMI_CFG_PAM_A1._402 := PPJ203.IN_ConfigPresent;

HMI_CFG_PAM_3._600 	:= TTJ[203].IN_ConfigPresent;
HMI_CFG_PAM_3._603	:= TTJ[203].IN_ConfigPresent;
HMI_CFG_PAM_3._604	:= TTJ[203].IN_ConfigPresent;
HMI_CFG_PAM_3._606 	:= LTJ[203].IN_ConfigPresent;
HMI_CFG_PAM_3._607 	:= LTJ[203].IN_ConfigPresent;
HMI_CFG_PAM_3._608 	:= LTJ[203].IN_ConfigPresent;
HMI_CFG_PAM_3._610	:= LTJ[203].IN_ConfigPresent;
HMI_CFG_PAM_3._611	:= PPJ203.IN_ConfigPresent;
HMI_CFG_PAM_3._612	:= PPJ203.IN_ConfigPresent;
HMI_CFG_PAM_3._613	:= AVJ[217].IN_ConfigPresent;
HMI_CFG_PAM_3._614	:= AVJ[217].IN_ConfigPresent;
HMI_CFG_PAM_3._615	:= PPJ[202].IN_ConfigPresent;
HMI_CFG_PAM_3._616	:= VAR_DOS_HotProductControl;
HMI_CFG_PAM_3._620	:= TTJ[203].IN_ConfigPresent;
HMI_CFG_PAM_3._621	:= TTJ[203].IN_ConfigPresent;
HMI_CFG_PAM_3._622	:= TRUE;
HMI_CFG_PAM_3._623	:= TRUE;
HMI_CFG_PAM_3._624	:= TRUE;
HMI_CFG_PAM_3._626	:= LTJ[203].IN_ConfigPresent;
HMI_CFG_PAM_3._630	:= PPJ[202].IN_ConfigPresent;
HMI_CFG_PAM_3._631	:= TRUE;
HMI_CFG_PAM_3._632	:= TRUE;
HMI_CFG_PAM_3._633	:= TTJ[203].IN_ConfigPresent;
HMI_CFG_PAM_3._634	:= PPJ203.IN_ConfigPresent;
HMI_CFG_PAM_3._635	:= PPJ203.IN_ConfigPresent;
HMI_CFG_PAM_3._636	:= AVJ[217].IN_ConfigPresent;
HMI_CFG_PAM_3._637	:= AVJ[217].IN_ConfigPresent;
HMI_CFG_PAM_3._640	:= FALSE;
HMI_CFG_PAM_3._641	:= TRUE;
HMI_CFG_PAM_3._642	:= TRUE;
HMI_CFG_PAM_3._643	:= TRUE;
HMI_CFG_PAM_3._644	:= FALSE;
HMI_CFG_PAM_3._645	:= TRUE;

HMI_CFG_PAM_D1._611	:= PPJ[202].IN_ConfigPresent;
HMI_CFG_PAM_D1._612	:= PPJ[202].IN_ConfigPresent;
HMI_CFG_PAM_D1._613	:= PPJ[202].IN_ConfigPresent;
HMI_CFG_PAM_D1._616	:= PPJ[202].IN_ConfigPresent;
HMI_CFG_PAM_D1._617	:= PPJ[202].IN_ConfigPresent;
HMI_CFG_PAM_D1._618	:= PPJ[202].IN_ConfigPresent;

HMI_CFG_PAC_1._015 := TRUE;
HMI_CFG_PAC_1._018 := TRUE;
HMI_CFG_PAC_1._025 := TRUE;
HMI_CFG_PAC_1._500 := TRUE;
HMI_CFG_PAC_1._501 := TRUE;
//HMI_CFG_PAC_1._502 := TRUE;
//HMI_CFG_PAC_1._503 := TRUE;
HMI_CFG_PAC_1._505 := TRUE;
HMI_CFG_PAC_1._510 := TRUE;
END_ACTION
TRANSITION PULP FROM DOS_Cfg TO (DOSVar,Instruments,ModeSelection,MainSequencer,Valves,Pumps,Motor,Lifting,DataTo):=
TRUE
END_TRANSITION
TRANSITION FLAVOR FROM DOS_Cfg TO DataToF:=
FALSE
END_TRANSITION
STEP DataToF:
DOS_DataOutFlavor; //RMH017
DOS_AlarmFlavor;
END_STEP
TRANSITION FROM DataToF TO DOSInit:=
FALSE
END_TRANSITION
(* @SFCISJUMP := 'DOSInit' *)
STEP DOSVar:
VAR_DOS_Blink1HzEp 		:= EDGEPOS(AID.DataOut.Blink1Hz);
VAR_DOS_PBResetEp		:= EDGEPOS(AID.DataOut.Reset);
VAR_DOS_HotProductControl := NOT CFG_Par.Machine.Type.SRMA;
END_STEP
STEP Instruments:
DOS_InstrTemp;
DOS_InstrLevel;
DOS_InstrVolume;
DOS_InstrPosition;
DOS_InstrPress;
DOS_InstrFlow;
END_STEP
STEP ModeSelection:
DOS_ModeSelection;
DOS_ManualLifting;
END_STEP
STEP MainSequencer:
DOS_StepManager;
DOS_StepMove;
DOS_StepConfig;
DOS_StepStatus;
END_STEP
STEP Valves:
DOS_ValvesLogic;
DOS_ValvesFlip;
DOS_ValvesFB;
DOS_ModulatingPID;
END_STEP
STEP Pumps:
DOS_PumpsLogic;
DOS_PumpsPID;
DOS_PumpsFB;
END_STEP
STEP Motor:
DOS_MotorsLogic;
DOS_MotorsFB;
END_STEP
STEP Lifting:
LiftMoveMngt_Doser;
END_STEP
STEP DataTo:
DOS_DataOut;
DOS_HMI;
DOS_Alarm;
END_STEP
TRANSITION FROM (DOSVar,Instruments,ModeSelection,MainSequencer,Valves,Pumps,Motor,Lifting,DataTo) TO DOS_Off:=
FALSE
END_TRANSITION
STEP DOS_Off:
ST_tmp_suspend(0);
END_STEP
TRANSITION FROM DOS_Off TO DOSInit:=
FALSE
END_TRANSITION
(* @SFCISJUMP := 'DOSInit' *)
END_PROGRAM
```

#### DOS_Devices.var - Local variables
```iecst
(*MOTORS*)
VAR
	MMF : ARRAY[MIN_CFG_AVx..MAX_CFG_AVx] OF Motor_FC280_Vfd;
	MMJ : ARRAY[MIN_CFG_AVx..MAX_CFG_AVx] OF Motor_FC280_Vfd;
	PPJ : ARRAY[MIN_CFG_AVx..MAX_CFG_AVx] OF Motor_FC280_Vfd;
	PPJ203 : Valve_Mod;
	PPJ203_AuxScale : LCRScal;
END_VAR
(*VALVES*)
VAR
	AVJ : ARRAY[MIN_CFG_AVx..MAX_CFG_AVx] OF Valve_Dig;
	PDO_YV65 : Valve_Dig;
	_211CPF : Valve_Dig;
	RVJ : ARRAY[MIN_CFG_RVx..MAX_CFG_RVx] OF Valve_Mod;
END_VAR
(*ANALOG*)
VAR
	TTJ : ARRAY[MIN_CFG_TTx..MAX_CFG_TTx] OF Analog_In;
	LTJ : ARRAY[MIN_CFG_LTx..MAX_CFG_LTx] OF Analog_In;
	_210PTF : Digital_Obj;
	_205MEF : Analog_In_Direct_Inverse;
	_206MEF : Analog_In_Direct_Inverse;
END_VAR
(*DIGITAL*)
VAR
	LSJ200L : Digital_Obj;
	LSJ200M : Digital_Obj;
	LSJ200H : Digital_Obj;
	LSJ : ARRAY[MIN_CFG_LSx..MAX_CFG_LSx] OF Digital_Obj;
	FSJ : ARRAY[MIN_CFG_FSx..MAX_CFG_FSx] OF Digital_Obj;
	_210DSX : Digital_Obj; (*Cop arm in cleaning position*)
	_211DSX : Digital_Obj; (*Cop arm in production pos*)
	_215DSF : Digital_Obj;
	_216DSF : Digital_Obj;
	_212DSF : Digital_Obj;
	_213DSF : Digital_Obj;
	_217DSF : Digital_Obj;
END_VAR
```

#### Variables.var - Local variables
```iecst
(*SELECTIONS*)
VAR
	VAR_DOS_FMDProduction : BOOL;
	VAR_DOS_FMDProductionFillerOnly : BOOL;
	VAR_DOS_FMDDrain : BOOL;
	VAR_DOS_FMDCip : BOOL;
	VAR_DOS_FMDRinse : BOOL;
	VAR_DOS_FMDCop : BOOL;
	VAR_DOS_FMDByPass : BOOL;
	VAR_DOS_FMDPositionRequest : BOOL;
	VAR_DOS_FMDPositioning : BOOL;
	VAR_DOS_MemPBStart : BOOL;
	VAR_DOS_MemPBStop : BOOL;
	VAR_DOS_MemPBAbort : BOOL;
	VAR_DOS_MemPBSkipForward : BOOL;
	VAR_DOS_MemSSPause : BOOL;
END_VAR
(*AUXILIARY VARIABLES*)
VAR
	VAR_DOS_Blink1HzEp : BOOL;
	VAR_DOS_PBResetEp : BOOL;
	VAR_DOS_HotProductControl : BOOL;
	VAR_DOS_InletOpen : BOOL;
	VAR_DOS_LoopOpen : BOOL;
	VAR_DOS_ReturnOpen : BOOL;
	VAR_DOS_RVJ201Auto : BOOL;
	VAR_DOS_SelectionLost : BOOL;
	VAR_DOS_BypassRequest : BOOL;
	VAR_DOS_TankEmpted : BOOL;
	VAR_DOS_LiftSelectionEnable : BOOL;
	VAR_DOS_SS2PSelectionEnable : BOOL;
	VAR_DOS_CleanArmProdPos : BOOL;
	VAR_DOS_CleanArmCopPos : BOOL;
	VAR_DOS_CleanArmCopPosFault : BOOL;
	VAR_DOS_SeqBackupAllowed : BOOL;
	VAR_DOS_RinseCycle : REAL;
	VAR_DOS_MotorReady : UINT;
	VAR_DOS_SeqFor : UINT;
	VAR_DOS_ForIndex : UINT;
	VAR_DOS_LevelPercentage : REAL;
	VAR_DOS_LevelVolume : REAL;
	VAR_DOS_LevelHeight : REAL;
END_VAR
(*ALARM VARIABLES*)
VAR
	VAR_DOS_WaterTemperatureTooHigh : BOOL;
	VAR_DOS_WaterTemperatureTooLow : BOOL;
	VAR_DOS_TankTooLow : BOOL;
	VAR_DOS_TankSafetyLimit : BOOL;
	VAR_DOS_TankTooFull : BOOL;
	VAR_DOS_AVJ_ValveFault : BOOL;
	VAR_DOS_MotorFault : BOOL;
	VAR_DOS_NoBotNoFillPressureLow : BOOL;
	VAR_DOS_NoBotNoFillPressureFault : BOOL;
END_VAR
(*AUXILIARY TIMERS*)
VAR
	TMR_TON_TemperatureTooLow : TON;
	TMR_TON_InletSafetyDelay : TON;
	TMR_TOF_FlipWork : ARRAY[0..2] OF TOF;
	TMR_TON_FlipWait : ARRAY[0..2] OF TON;
END_VAR
(*SAFETY STATUS*)
VAR
	VAR_DOS_ValveEnable : BOOL;
	VAR_DOS_PumpEnable : BOOL;
	VAR_DOS_AlarmActive : BOOL;
	VAR_DOS_MotorEnable : BOOL;
END_VAR
(*PID*)
VAR CONSTANT
	PID_MODE_CIP : USINT := 0;
	PID_MODE_PRD : USINT := 1;
END_VAR
VAR
	FB_PID_PPJ202 : ARRAY[0..3] OF PID_Cont;
	FB_PID_RVJ201 : ARRAY[0..3] OF PID_Cont;
END_VAR
(*Manual Lifting*)
VAR
	VAR_DOS_MoveInProductionPosition : USINT;
	VAR_DOS_MoveInCOPPosition : USINT;
	VAR_DOS_MoveInCIPPosition : USINT;
END_VAR
```

#### VariablesSeq.var - Local variables
```iecst
(*SEQUENCER*)
VAR
	FB_DOS_SEQ : Sequencer_v2;
	VAR_DOS_SEQ_Step : SEQ_Type;
	VAR_DOS_Lift_SEQ_Step : SEQ_Type;
	VAR_DOS_Lift_SEQ : SEQ_Module_Type;
	VAR_DOS_SEQ : SEQ_Module_Type;
	VAR_DOS_SeqProdStopAlarm : BOOL;
	VAR_DOS_SeqProdStopRequest : BOOL;
	VAR_DOS_SeqProdAbortRequest : BOOL;
	VAR_DOS_SeqCipStopAlarm : BOOL;
	VAR_DOS_SeqRinseStopAlarm : BOOL;
	VAR_DOS_SeqRinseStopRequest : BOOL;
	VAR_DOS_SeqCipStopRequest : BOOL;
	VAR_DOS_SeqRinseAbortRequest : BOOL;
	VAR_DOS_SeqCipAbortRequest : BOOL;
	VAR_DOS_SeqDrainStopAlarm : BOOL;
	VAR_DOS_SeqDrainStopRequest : BOOL;
	VAR_DOS_SeqDrainAbortRequest : BOOL;
	VAR_DOS_SeqBypassStopAlarm : BOOL;
	VAR_DOS_SeqBypassAbortRequest : BOOL;
	VAR_DOS_SeqPositionRequest : BOOL;
	VAR_DOS_SeqPositionReached : BOOL;
	VAR_index : UINT;
	VAR_DOS_SeqActualStep : UINT;
	VAR_DOS_SeqCyclesCounter : UDINT;
END_VAR
(*MODE VARIABLES*)
VAR
	VAR_DOS_ModeWait : BOOL;
	VAR_DOS_ModeProduction : BOOL;
	VAR_DOS_ModeProductionExcluded : BOOL;
	VAR_DOS_ModeCip : BOOL;
	VAR_DOS_ModeRinse : BOOL;
	VAR_DOS_ModeDrain : BOOL;
	VAR_DOS_ModeCop : BOOL;
	VAR_DOS_ModePositionRequest : BOOL;
	VAR_DOS_ModePositioning : BOOL;
	VAR_DOS_ModeBypass : BOOL;
	VAR_DOS_MemProdDrain : BOOL;
	VAR_DOS_MemWaitPumpSet : BOOL;
	VAR_DOS_ModeWaitOperator : BOOL;
	VAR_DOS_MemDoserByPassed : BOOL;
	VAR_DOS_MemDoserIncluded : BOOL;
	VAR_DOS_MemDoserAxisOff : BOOL;
	VAR_DOS_MemDoserAxisOn : BOOL;
	VAR_DOS_MemFillerAxisOffReq : BOOL;
	VAR_DOS_PhasingWithDos : BOOL;
	VAR_DOS_PhasingWithoutDos : BOOL;
END_VAR
(*STEP VARIABLES*)
(*Production*)
VAR
	VAR_DOS_StepProdHeating : BOOL;
	VAR_DOS_StepProdProducing : BOOL;
	VAR_DOS_StepProdLowLevel : BOOL;
	VAR_DOS_StepProdRecovery : BOOL;
	VAR_DOS_StepProdStopped : BOOL;
	VAR_DOS_StepProdAborted : BOOL;
END_VAR
(*Cip*)
VAR
	VAR_DOS_StepCipCleaning : BOOL;
	VAR_DOS_StepCipDraining : BOOL;
	VAR_DOS_StepCipRecovery : BOOL;
	VAR_DOS_StepCipStopped : BOOL;
	VAR_DOS_StepCipAborted : BOOL;
	VAR_DOS_StepCipFillerStartEnable : BOOL;
	VAR_DOS_StepCipEnded : BOOL;
END_VAR
(*Rinse*)
VAR
	VAR_DOS_StepRinseReq : BOOL;
	VAR_DOS_StepRinseInExecution : BOOL;
	VAR_DOS_StepRinseStopped : BOOL;
	VAR_DOS_StepRinseAborted : BOOL;
END_VAR
(*Drain*)
VAR
	VAR_DOS_StepDrainStopped : BOOL;
	VAR_DOS_StepDrainAborted : BOOL;
END_VAR
(*Cop*)
VAR
	VAR_DOS_StepCopRunning : BOOL;
END_VAR
(*FLIP SEQUENCE*)
VAR CONSTANT
	VAR_DOS_FlipSeqMax : USINT := 10;
END_VAR
VAR
	VAR_DOS_FlipIndex : USINT;
	VAR_DOS_FlipSequenceRepetition : USINT;
	VAR_DOS_Flip_CycleTime : REAL;
	VAR_DOS_FlipSeqStart : BOOL;
	VAR_DOS_FlipSeqEnable : BOOL;
	VAR_DOS_FlipSeqReset : BOOL;
	VAR_DOS_FlipSeqEnd : BOOL;
	VAR_DOS_FlipSeqValve : ARRAY[0..VAR_DOS_FlipSeqMax] OF DOS_ValveFlip_Type;
END_VAR
(*PRODUCTION END*)
VAR
	VAR_DOS_ProdEndRequest : {REDUND_UNREPLICABLE} BOOL;
	VAR_DOS_StepProdEndProduction : {REDUND_UNREPLICABLE} BOOL;
	VAR_DOS_EndProdStopContainer : {REDUND_UNREPLICABLE} BOOL;
	VAR_DOS_RejectExpulsionRequest : {REDUND_UNREPLICABLE} BOOL;
	VAR_DOS_ProdEndRejectContainers : {REDUND_UNREPLICABLE} REAL;
	VAR_DOS_ProdEndAvailableLiters : {REDUND_UNREPLICABLE} REAL;
	VAR_DOS_ProdEndNecessaryLiters : {REDUND_UNREPLICABLE} REAL;
	VAR_DOS_ProdEndNecessaryBottle : {REDUND_UNREPLICABLE} REAL; (*v999hema*)
END_VAR
(*By Pass*)
VAR
	VAR_DOS_StepCamPositioning : BOOL;
	VAR_DOS_StepCamPosInProgress : BOOL;
	VAR_DOS_StepCamPosRequest : BOOL;
	VAR_DOS_StepBypassAborted : BOOL;
END_VAR
(*Motion*)
VAR
	VAR_DOS_StepMotorization : BOOL;
	VAR_DOS_Flip_RTInfo : RTInfo;
END_VAR
```

#### Types.typ - Local data types
```iecst
TYPE
	SEQ_Type : 	STRUCT
		Step : ARRAY[0..MAX_STEP_CFG]OF SEQ_Step_Type;
		ModeActual : UINT;
		StepActual : UINT;
		TON_Time_END : BOOL;
		T_Time_END : BOOL;
		TO_Time_END : BOOL;
		Laps_Done : BOOL;
		Cycles_Done : BOOL; (*All Cycles Done*)
	END_STRUCT;
	SEQ_Step_Type : 	STRUCT
		Jump : ARRAY[0..MAX_JUMP_CFG]OF SEQ_Jump_Type;
		Config : SEQ_StepConfig_Type;
	END_STRUCT;
	SEQ_Jump_Type : 	STRUCT
		Condition : BOOL;
		Number : UINT;
	END_STRUCT;
	ActionReq_Type : 	STRUCT
		Req : BOOL;
		Done : BOOL;
	END_STRUCT;
END_TYPE

(*DEVICES*)

TYPE
	SEQ_Module_Type : 	STRUCT
		Device : SEQ_Device_Type;
		Mem : SEQ_Mem_Type;
		ITC : SEQ_Itc_Type;
	END_STRUCT;
	SEQ_Mem_Type : 	STRUCT
		ContainersStop : BOOL; (*Containers Stop Control (1 = Stop)*)
		MachineStart : BOOL;
		MachineStop : BOOL;
		DummyBottles : BOOL; (*Dummy Bottle Install*)
		PositioningRequest : BOOL; (*Request of Cam Positioning at height SP of Sequncer*)
		COP_Cycle : BOOL; (*Cycle of COP Active*)
		DosingOn : BOOL; (*Dosing*)
		LapsCounter : BOOL; (*Laps Conter Req*)
		ValveOpening : BOOL;
		CopAfterCipRequest : BOOL; (*Request of COP after CIP end*)
		PBAbortEnable : BOOL; (*PB Abort Sequence Enable*)
		PBStopEnable : BOOL; (*PB Stop Sequence Enable*)
		PBStartEnable : BOOL; (*PB Start Sequence Enable*)
	END_STRUCT;
	SEQ_Device_Type : 	STRUCT
		AVJ201 : Valve_Cmd_Type;
		AVJ210 : Valve_Cmd_Type;
		AVJ211 : Valve_Cmd_Type;
		AVJ212 : Valve_Cmd_Type;
		AVJ215 : Valve_Cmd_Type;
		AVJ216 : Valve_Cmd_Type;
		AVJ217 : Valve_Cmd_Type;
		AVJ218 : Valve_Cmd_Type;
		AVJ221 : Valve_Cmd_Type;
		AVJ230 : Valve_Cmd_Type;
		AVJ231 : Valve_Cmd_Type;
		AVJ232 : Valve_Cmd_Type;
		AVJ233 : Valve_Cmd_Type;
		AVJ234 : Valve_Cmd_Type;
		AVJ235 : Valve_Cmd_Type;
		RVJ201_PID : PID_Type;
		PPJ201_PID : PID_Type;
		PPJ202_PID : PID_Type;
		PPJ203_PID : PID_Type;
		MMJ201_PID : PID_Type;
		LSJ200 : Digital_In_Type;
		LSJ201 : Digital_In_Type;
		LSJ202 : Digital_In_Type;
		FSJ201 : Digital_In_Type;
		FSJ202 : Digital_In_Type;
		LTJ203 : Analog_In_Type;
		TTJ203 : Analog_In_Type;
	END_STRUCT;
	SEQ_Itc_Type : 	STRUCT
		CIP_CleaningMode : BOOL; (*To CIP -> Filler in Mode Cip*)
		CIP_CleaningRequest : BOOL; (*To CIP -> Request of Solution Sending*)
		CIP_Alarm : BOOL; (*To CIP -> Critical Alarm Present*)
		CIP_RinseEnded : BOOL; (*To CIP -> Rinse Finished*)
		CIP_ChangeEnded : BOOL; (*To CIP -> Change Finished*)
		CIP_DrainRunning : BOOL; (*To CIP -> Drain Cycle Running*)
		CIP_RinseRunning : BOOL; (*To CIP -> Rinse Cycle Running*)
		CIP_CleaningRunning : BOOL; (*To CIP -> Cleaning Cycle Running*)
		CIP_DrainEnded : BOOL; (*To CIP -> Drain Finished*)
		CIP_FloodingEnded : BOOL; (*To CIP -> Drain Finished*)
		CIP_FlipEnable : BOOL; (*To CIP -> Drain Finished*)
		CIP_CycleEnded : BOOL; (*To CIP -> Drain Finished*)
		PROD_ReadyForHeating : BOOL; (*To PASTO-> Filler Ready for Production (Heating)*)
		PROD_DoserInTemperature : BOOL; (*To PASTO-> Filler Temperature OK (After Heating)*)
		PROD_ProductRequest : BOOL; (*To PASTO-> Product Request *)
		PROD_DoserOnFillingMode : BOOL; (*To PASTO-> Product Consumend -Filling Valve Opening*)
		PROD_EndProductionCompleted : BOOL; (*To PASTO-> End Production Done*)
		PROD_ProductRecoveryEnd : BOOL; (*To PASTO-> Product Recovery End*)
		PROD_WaterRequestAfterProd : BOOL; (*To PASTO-> Water Request For Filler Rinse Afetr Production*)
	END_STRUCT;
	Analog_In_Type : 	STRUCT
		ALR_HighLimitEn : BOOL;
		ALR_HighLimitSP : REAL;
		ALR_LowLimitEn : BOOL;
		ALR_LowLimitSP : REAL;
		SP : REAL;
		CMP : USINT;
		MinDev : REAL;
		MaxDev : REAL;
	END_STRUCT;
	Digital_In_Type : 	STRUCT
		ALR : BOOL;
		WAIT_ON : BOOL;
		WAIT_OFF : BOOL;
	END_STRUCT;
	PID_Type : 	STRUCT
		PID_Enable : BOOL; (*PID Enable Condition*)
		PID_Mode : BOOL; (*PID Mode (1 = Auto - 0 = Manual)*)
		Auto_SP_Value : REAL;
		Auto_SP_MinDev : REAL;
		Auto_SP_MaxDev : REAL;
		FIX_Value : REAL;
	END_STRUCT;
	Valve_Cmd_Type : 	STRUCT
		AutoCnd : BOOL;
		EnableCnd : BOOL;
		FlipGroup : UINT;
	END_STRUCT;
	Motor_Cmd_Type : 	STRUCT
		AutoCnd : BOOL;
	END_STRUCT;
	DOS_ValveFlip_Type : 	STRUCT
		Config : BOOL; (*Flip Sequence Configured*)
		Request : BOOL; (*Flip Sequence Request to Valve*)
		Executed : BOOL; (*Flip Sequence Done by Valve*)
		Done : BOOL; (*Flip Sequence Done Memory*)
		SequenceDone : BOOL; (*Flip Sequence Completed*)
		TimeDelay_SP : REAL; (*Next Flip Sequence Delay*)
		TimeDelay_PV : REAL; (*Next Flip Sequence Delay Elapsed*)
	END_STRUCT;
END_TYPE
```

#### DOS_Lifting.var - Local variables
```iecst
VAR
	VAR_DOS_Lift_State : VAR_DOS_LiftCommands_Type;
	VAR_DOS_MMF205 : VAR_DOS_MMF205_Type;
	VAR_DOS_MMF206 : VAR_DOS_MMF206_Type;
	FbLCRLimScal_ml_mm : LCRLimScal;
	FbLCRLimScal_mm_ml : LCRLimScal;
	VAR_DOS_PistonVolume_ml : REAL;
	VAR_DOS_PistonVolume_mm : REAL;
	ml : USINT := 1;
	mm : USINT := 0;
END_VAR
(*Check lifting - ALARM*)
VAR
	TON_DosRunFbk : ARRAY[0..1] OF TON;
	VAR_MMF205PositionSave : REAL;
	VAR_MMF206PositionSave : REAL;
	VAR_MMF205Down : BOOL;
	VAR_MMF206Down : BOOL;
	TON_DosPositionCheck : ARRAY[0..1] OF TON;
	VAR_OldMMF205Position : REAL;
	VAR_OldMMF206Position : REAL;
	VAR_MMF205DirectionReverse : BOOL;
	VAR_MMF206DirectionReverse : BOOL;
END_VAR
```

#### DOS_Lifting.typ - Local data types
```iecst
TYPE
	VAR_DOS_LiftCommands_Type : 	STRUCT
		Position : VAR_DOS_Position_Type;
		DevicesDetails : VAR_DOS_DevicesDetails_Type;
		WarningsDetails : VAR_DOS_Warnings_Type;
		CmdSizeChangeHeight : VAR_DOS_CmdHeight_Type;
		CmdProductionHeight : VAR_DOS_CmdProductionHeight_Type;
		CmdMaxHeight : VAR_DOS_CmdMaxHeight_Typ;
		CmdCipHeight : VAR_DOS_CmdCipHeight_Typ;
		CmdManualMode : VAR_DOS_CmdManualMode_Type;
		DevicesGeneralAlarm : BOOL;
		CaruselPositioning : BOOL;
		MachineStopReq : BOOL;
		StepActual : USINT;
		ChangeOver : USINT;
	END_STRUCT;
	VAR_DOS_Position_Type : 	STRUCT
		ActualSp : REAL;
		ActualPv : REAL;
		MinMechanicalHeight : REAL;
		MinMechanicalHeightReached : BOOL;
		MaxMechanicalHeight : REAL;
		MaxMechanicalHeightReached : BOOL;
	END_STRUCT;
	VAR_DOS_DevicesDetails_Type : 	STRUCT
		IsolatedAlr : BOOL;
		ContactorFbkAlr : BOOL;
		BrakePositionAlr : BOOL;
		ProbeAlr : BOOL;
		DirectionAlr : BOOL;
		RunFbkAlr : BOOL;
		OverloadAlr : BOOL;
		ContactorAlr : BOOL;
		ShaftBrokenAlr : BOOL;
	END_STRUCT;
	VAR_DOS_Warnings_Type : 	STRUCT
		OutOfPosition : BOOL;
	END_STRUCT;
	VAR_DOS_CmdHeight_Type : 	STRUCT
		Req : BOOL;
		Done : BOOL;
	END_STRUCT;
	VAR_DOS_CmdProductionHeight_Type : 	STRUCT
		Req : BOOL;
		Sp : REAL;
		Done : BOOL;
	END_STRUCT;
	VAR_DOS_CmdMaxHeight_Typ : 	STRUCT
		Req : BOOL;
		Sp : REAL;
		Done : BOOL;
	END_STRUCT;
	VAR_DOS_CmdCipHeight_Typ : 	STRUCT
		Req : BOOL;
		Sp : REAL;
		Done : BOOL;
	END_STRUCT;
	VAR_DOS_CmdManualMode_Type : 	STRUCT
		Req : BOOL;
		Up : BOOL;
		Dwn : BOOL;
		UpperLimitReached : BOOL;
		LowerLimitReached : BOOL;
	END_STRUCT;
	VAR_DOS_MMF205_Type : 	STRUCT  (*Motor Lifting *)
		PosValid : BOOL;
		SensorMaxVol : BOOL;
		SensorHighPos : BOOL;
		SensorLowPos : BOOL;
		PosReached : BOOL;
		PosActual : ARRAY[0..1]OF REAL;
		SpActual : ARRAY[0..1]OF REAL;
	END_STRUCT;
	VAR_DOS_MMF206_Type : 	STRUCT
		PosValid : BOOL;
		PosOffset : BOOL;
		SensorHighPos : BOOL;
		SensorLowPos : BOOL;
		PosReached : BOOL;
		PosActual : ARRAY[0..1]OF REAL;
		SpActual : ARRAY[0..1]OF REAL;
	END_STRUCT;
	VAR_DOS_LimitsExceeded_Type : 	STRUCT  (*Mom uso?*)
		UpperLimitExceededAlr : BOOL;
		LowerLimitExceededAlr : BOOL;
	END_STRUCT;
	VAR_DOS_ChangeOverData_Type : 	STRUCT  (*non uso?*)
		ChangeOverNecessary : BOOL;
		ActualFormatHeight : ARRAY[0..5]OF REAL;
		RecipeFormatHeight : ARRAY[0..5]OF REAL;
	END_STRUCT;
END_TYPE
```

#### DOS_Lift_Sequencer.var - Local variables
```iecst
VAR
	VAR_DOS_LiftStepMem : VAR_DOS_LiftMoveStep_Type;
	VAR_DOS_LiftMMF206SeqMem : VAR_DOS_LiftSeqMem_Type;
	VAR_DOS_LiftMMF205SeqMem : VAR_DOS_LiftSeqMem_Type;
	VAR_DOS_LiftMoveStep : VAR_DOS_LiftMoveStep_Type;
END_VAR
```

#### DOS_Lift_Sequencer.typ - Local data types
```iecst
TYPE
	VAR_DOS_LiftMoveStep_Type :
		(
		DSR_LiftSystemOff,
		DSR_ProbeZeroReq,
		DSR_ProbeZeroLowPos,
		DSR_ProbeZeroDisengSensLow,
		DSR_ProbeZeroWaitSensLowPos,
		DSR_ProbeZeroDone,
		DSR_CopPosReached,
		DSR_DosingReq,
		DSR_DosingActive,
		DSR_Manual,
		DSR_PosMMF206ToMMF205,
		DSR_UpMMF205andMMF206,
		DSR_DwnMMF205andMMF206,
		DSR_PosReached,
		DSR_Fault
		);
	VAR_DOS_LiftSeqMem_Type : 	STRUCT
		Unlock : BOOL;
		LiftMotor : VAR_DOS_SeqMemLiftMotor_Type;
		Position : VAR_DOS_SeqMemPosition_Type;
		Sensor : VAR_DOS_SeqMemSensor_Type;
	END_STRUCT;
	VAR_DOS_SeqMemLiftMotor_Type : 	STRUCT
		Up : BOOL;
		Dwn : BOOL;
		RunFbkAlr : BOOL;
		DirectionAlr : BOOL;
	END_STRUCT;
	VAR_DOS_SeqMemPosition_Type : 	STRUCT
		ActualSp : REAL;
		SizeChangeHeightReached : BOOL;
		ProductionHeightReached : BOOL;
		MaxMechanicalHeightReached : BOOL;
		ManUpperLimitReached : BOOL;
		ManLowerLimitReached : BOOL;
	END_STRUCT;
	VAR_DOS_SeqMemSensor_Type : 	STRUCT
		SensorMaxVolWaitOff : BOOL;
		SensorLowPosWaitOn : BOOL;
		SensorHighPosWaitOn : BOOL;
		SensorLowPosWaitOff : BOOL;
		SensorHighPosWaitOff : BOOL;
		SensorMaxVolWaitOn : BOOL;
	END_STRUCT;
END_TYPE
```

#### Structures.var
```iecst
(*//Lift position Selection ComboBox*)
VAR
	VAR_LiftPositionType : DOS_Lift_Phase_Type;
END_VAR
```

#### Structures.typ
```iecst
TYPE
	DOS_Lift_Phase_Type : 	STRUCT
		Elements : ARRAY[0..19]OF HMI_ComboBoxElements_Type; (*vrma*)
		Data : ARRAY[0..19]OF DOS_LiftPhase_Type;
	END_STRUCT;
	DOS_LiftPhase_Type : 	STRUCT
		PhaseType : USINT;
	END_STRUCT;
END_TYPE
```

#### DOS_InstrTemp.st
```iecst
ACTION DOS_InstrTemp:

	TTJ[203](
	IN_ConfigPresent 	:= TTJ[203].IN_ConfigPresent,
	IN_FaultOutMode 	:= CST_AI_FaultMode_High,
	IN_EngScale 		:= TTJ[203].IN_EngScale,
	IN_CompareMode 		:= VAR_DOS_SEQ.Device.TTJ203.CMP,
	IN_AlarmEn 			:= TRUE,
	IN_MaskEn 			:= TRUE,
	IN_Reset 			:= VAR_DOS_PBResetEp,
	IN_ActualSP 		:= VAR_DOS_SEQ.Device.TTJ203.SP, //INT_TO_REAL(PstFlr.SPTemp / 10)  o quel segnale è solo in CIP il SetPoint? FILIPPO
	IN_MinDev 			:= VAR_DOS_SEQ.Device.TTJ203.MinDev,
	IN_MaxDev 			:= VAR_DOS_SEQ.Device.TTJ203.MaxDev,
	IN_WaitDelay 		:= T#500ms,
	IN_HighLimitEn 		:= VAR_DOS_SEQ.Device.TTJ203.ALR_HighLimitEn,
	IN_HighLimitSP 		:= VAR_DOS_SEQ.Device.TTJ203.ALR_HighLimitSP,
	IN_HighLimitHyst 	:= 3.0,
	IN_HighLimitDelay 	:= T#3s,
	IN_LowLimitEn 		:= VAR_DOS_SEQ.Device.TTJ203.ALR_LowLimitEn,
	IN_LowLimitSP 		:= VAR_DOS_SEQ.Device.TTJ203.ALR_LowLimitSP,
	IN_LowLimitHyst 	:= 3,
	IN_LowLimitDelay 	:= T#3s,
	IN_TotPulseWeight 	:= 0.0,
	IN_TotType 			:= 0,
	IN_PLCCounterEn 	:= FALSE,
	IN_PLCCounterSP 	:= 0.0,
	IN_PLCCounterReset	:= FALSE,
	IN_HMITotEn 		:= FALSE,
	IN_HMITotReset 		:= FALSE,
	IO 					:= IO_TTJ[203],
	HMI 				:= HMI_TTJ[203]
	);

	TMR_TON_TemperatureTooLow.IN := TTJ[203].OUT_LowLimit;
	TMR_TON_TemperatureTooLow.PT := T#20S;
	TMR_TON_TemperatureTooLow();

	//VAR_DOS_ChillingRequest			:= VAR_DOS_SEQ.Device.TTJ[203].CMP>0 AND NOT TTJ[203].OUT_SpReached AND NOT TTJ[203].OUT_LowLimit;
	VAR_DOS_WaterTemperatureTooHigh	:= TTJ[203].OUT_HighLimit;
	VAR_DOS_WaterTemperatureTooLow	:= TMR_TON_TemperatureTooLow.Q;

END_ACTION
```

#### DOS_InstrLevel.st
```iecst
ACTION DOS_InstrLevel:
//LTJ203
//	TMR_TON_PrepTankLowLimitDelay.IN 	:= VAR_CTP_SEQ.Device.LTB201.ALR_LowLimitEn;
//	TMR_TON_PrepTankLowLimitDelay.PT	:= T#5s;
//	TMR_TON_PrepTankLowLimitDelay();
//
//	IF TMR_TON_PrepTankLowLimitDelay.Q THEN
//		LTB[201].IN_LowLimitDelay := T#1s;
//	ELSE
//		LTB[201].IN_LowLimitDelay := T#5s;
//	END_IF

	LTJ[203](
	IN_ConfigPresent 	:= LTJ[203].IN_ConfigPresent,
	IN_FaultOutMode 	:= CST_AI_FaultMode_High,
	IN_EngScale 		:= LTJ[203].IN_EngScale,
	IN_CompareMode 		:= VAR_DOS_SEQ.Device.LTJ203.CMP,
	IN_AlarmEn 			:= TRUE,
	IN_MaskEn 			:= TRUE,
	IN_Reset 			:= VAR_DOS_PBResetEp,
	IN_ActualSP 		:= VAR_DOS_SEQ.Device.LTJ203.SP,
	IN_MinDev 			:= HMI_PAM_3._610,
	IN_MaxDev 			:= HMI_PAM_3._610,
	IN_WaitDelay 		:= T#500ms,
	IN_HighLimitEn 		:= VAR_DOS_SEQ.Device.LTJ203.ALR_HighLimitEn,
	IN_HighLimitSP 		:= VAR_DOS_SEQ.Device.LTJ203.ALR_HighLimitSP,
	IN_HighLimitHyst 	:= 5.0,
	IN_HighLimitDelay 	:= T#1s,
	IN_LowLimitEn 		:= VAR_DOS_SEQ.Device.LTJ203.ALR_LowLimitEn,
	IN_LowLimitSP 		:= VAR_DOS_SEQ.Device.LTJ203.ALR_LowLimitSP,
	IN_LowLimitHyst 	:= 5.0,
	IN_LowLimitDelay 	:= T#1s,
	IN_TotPulseWeight 	:= 0.0,
	IN_TotType 			:= 0,
	IN_PLCCounterEn 	:= FALSE,
	IN_PLCCounterSP 	:= 0.0,
	IN_PLCCounterReset	:= FALSE,
	IN_HMITotEn 		:= FALSE,
	IN_HMITotReset 		:= FALSE,
	IO 					:= IO_LTJ[203],
	HMI 				:= HMI_LTJ[203]
	);

	IF LTJ[203].OUT_LowLimit THEN
		VAR_DOS_TankTooLow		:= TRUE;
	ELSIF VAR_DOS_PBResetEp THEN
		VAR_DOS_TankTooLow		:= FALSE;
	END_IF

	IF LTJ[203].OUT_ActValue < 3.0 THEN
		VAR_DOS_TankSafetyLimit	:= TRUE;
	ELSIF LTJ[203].OUT_ActValue > 5.0 THEN
		VAR_DOS_TankSafetyLimit	:= FALSE;
	END_IF

	VAR_DOS_TankTooFull := LTJ[203].OUT_HighLimit;
	VAR_DOS_TankEmpted := LTJ[203].OUT_ActValue < 3; //PER STEPMOVE

	//TANK LEVEL CONTROL
	//CONVERTION TO %,liters,mm v000 : QUA CAMBIA LA STRUTTURA MULTI SCALE COME QUELLA CTF.CHIEDI A HMI
	FB_DOS_Data.IN_ConfigPresent			:= TRUE;
	FB_DOS_Data.IN_Wait						:= HMI_LTJ[203].Wait;
	FB_DOS_Data.IN_Sp_Type					:= FB_DOS_Data.IN_Sp_Type;
	FB_DOS_Data.IN_TNK_PV					:= LTJ[203].OUT_ActValue;
	FB_DOS_Data.IN_TNK_Diameter_mm			:= 540.0;
	FB_DOS_Data.IN_TNK_Bottom_liters		:= 10; //volume of Hema Tank [L]
	FB_DOS_Data.IN_ProbeLength_mm			:= 1000.0; //lenght of the tank level probe [mm] (680.0 mm la sonda ma Tank alto 1000mm)
	FB_DOS_Data.IN_FromFloor_ToZeroProbe_mm	:= 0.0; //Height From Floor To Zero Point Of The Level Probe [mm]
	FB_DOS_Data.IN_Scale[0].ActualSP		:= VAR_DOS_SEQ.Device.LTJ203.SP;

	FB_DOS_Data(HMI := HMI_DOS_Data);

	VAR_DOS_LevelPercentage := FB_DOS_Data.OUT_Scale[0].ActValue; //%
	VAR_DOS_LevelVolume		:= FB_DOS_Data.OUT_Scale[1].ActValue; //LITERS
	VAR_DOS_LevelHeight		:= FB_DOS_Data.OUT_Scale[2].ActValue; //mm

	//END OF PRODUCTION
	VAR_DOS_ProdEndNecessaryLiters 	:= (INT_TO_REAL(FlrSkd.ContainersInMachine) * HMI_PAR_1._215) / 1000.0;
	VAR_DOS_ProdEndAvailableLiters 	:= INT_TO_REAL(PstFlr.ProductAvailableLiters) + VAR_DOS_LevelVolume;
	VAR_DOS_ProdEndNecessaryBottle	:= VAR_DOS_ProdEndAvailableLiters / (HMI_PAR_1._215/1000);

	VAR_DOS_ProdEndRequest			:= VAR_DOS_MemPBStop OR PstFlr.EndProductionReq OR VAR_DOS_StepProdEndProduction;

	IF VAR_DOS_ProdEndRequest THEN
		IF VAR_DOS_ProdEndAvailableLiters <= VAR_DOS_ProdEndNecessaryLiters OR VAR_DOS_ProdEndAvailableLiters < 20.0 THEN
			VAR_DOS_EndProdStopContainer := TRUE;
		END_IF
	ELSE
		VAR_DOS_EndProdStopContainer := FALSE;
	END_IF

	//CONTROL ON BOTTLES IN TRANSIT OVER AVAILABLE LITERS
	IF EDGEPOS(VAR_DOS_EndProdStopContainer)THEN
		VAR_DOS_ProdEndRejectContainers := (ABS (VAR_DOS_ProdEndAvailableLiters - VAR_DOS_ProdEndNecessaryLiters)/(HMI_PAR_1._215/1000.0));
	END_IF

	//CONTROL ON INLET CLOSING AND PRODUCT AVAILABLE
	IF FlrSkd.ContainersInMachine>0 THEN
		VAR_DOS_RejectExpulsionRequest := VAR_DOS_ProdEndRejectContainers > FlrSkd.ContainersInMachine;
	ELSE
		VAR_DOS_RejectExpulsionRequest 	:= FALSE;
		VAR_DOS_ProdEndRejectContainers	:= 0.0;
	END_IF

//LSJ200
	LSJ200L(
	IN_ConfigPresent 	:= LSJ200L.IN_ConfigPresent,
	IN_Alarm 			:= FALSE,
	IN_AlarmOnReq		:= LSJ200L.IN_WaitOff,
	IN_AlarmOffReq 		:= LSJ200L.IN_WaitOn,
	IN_SwitchDelay 		:= T#500ms,
	IN_WaitOn 			:= FALSE,
	IN_WaitOff 			:= FALSE,
	IN_OnDelay			:= T#5s,
	IN_OffDelay			:= T#5s,
	IN_Reset	 		:= VAR_DOS_PBResetEp,
	IN_MaskEn 			:= TRUE,
	IO 					:= IO_LSJ200L,
	HMI 				:= HMI_LSJ200L
	);

	LSJ200M(
	IN_ConfigPresent 	:= LSJ200M.IN_ConfigPresent,
	IN_Alarm 			:= FALSE,
	IN_AlarmOnReq		:= LSJ200M.IN_WaitOff,
	IN_AlarmOffReq 		:= LSJ200M.IN_WaitOn,
	IN_SwitchDelay 		:= T#500ms,
	IN_WaitOn 			:= FALSE,
	IN_WaitOff 			:= FALSE,
	IN_OnDelay			:= T#5s,
	IN_OffDelay			:= T#5s,
	IN_Reset	 		:= VAR_DOS_PBResetEp,
	IN_MaskEn 			:= TRUE,
	IO 					:= IO_LSJ200M,
	HMI 				:= HMI_LSJ200M
	);

	LSJ200H(
	IN_ConfigPresent 	:= LSJ200H.IN_ConfigPresent,
	IN_Alarm 			:= FALSE,
	IN_AlarmOnReq		:= LSJ200H.IN_WaitOff,
	IN_AlarmOffReq 		:= LSJ200H.IN_WaitOn,
	IN_SwitchDelay 		:= T#500ms,
	IN_WaitOn 			:= FALSE,
	IN_WaitOff 			:= FALSE,
	IN_OnDelay			:= T#5s,
	IN_OffDelay			:= T#5s,
	IN_Reset	 		:= VAR_DOS_PBResetEp,
	IN_MaskEn 			:= TRUE,
	IO 					:= IO_LSJ200H,
	HMI 				:= HMI_LSJ200H
	);

//LSJ201
	LSJ[201](
	IN_ConfigPresent 	:= LSJ[201].IN_ConfigPresent,
	IN_Alarm 			:= VAR_DOS_SEQ.Device.LSJ201.ALR,
	IN_AlarmOnReq		:= LSJ[201].IN_WaitOff,
	IN_AlarmOffReq 		:= LSJ[201].IN_WaitOn,
	IN_SwitchDelay 		:= T#500ms,
	IN_WaitOn 			:= VAR_DOS_SEQ.Device.LSJ201.WAIT_ON,
	IN_WaitOff 			:= VAR_DOS_SEQ.Device.LSJ201.WAIT_OFF,
	IN_OnDelay			:= T#5s,
	IN_OffDelay			:= T#5s,
	IN_Reset	 		:= VAR_DOS_PBResetEp,
	IN_MaskEn 			:= TRUE,
	IO 					:= IO_LSJ[201],
	HMI 				:= HMI_LSJ201H
	);

//LSJ202
	LSJ[202](
	IN_ConfigPresent 	:= LSJ[202].IN_ConfigPresent,
	IN_Alarm 			:= VAR_DOS_SEQ.Device.LSJ202.ALR,
	IN_AlarmOnReq		:= LSJ[202].IN_WaitOff,
	IN_AlarmOffReq 		:= LSJ[202].IN_WaitOn,
	IN_SwitchDelay 		:= T#500ms,
	IN_WaitOn 			:= VAR_DOS_SEQ.Device.LSJ202.WAIT_ON,
	IN_WaitOff 			:= VAR_DOS_SEQ.Device.LSJ202.WAIT_OFF,
	IN_OnDelay			:= T#5s,
	IN_OffDelay			:= T#5s,
	IN_Reset	 		:= VAR_DOS_PBResetEp,
	IN_MaskEn 			:= TRUE,
	IO 					:= IO_LSJ[202],
	HMI 				:= HMI_LSJ202H
	);
END_ACTION
```

#### DOS_InstrPosition.st
```iecst
ACTION DOS_InstrPosition:
//HDP UP Limit M5
	_215DSF(
	IN_ConfigPresent 	:= _215DSF.IN_ConfigPresent,
	IN_OnDelay			:= T#1s,
	IN_OffDelay			:= T#1s,
	IN_SwitchDelay		:= T#1s,
	IN_Reset	 		:= VAR_DOS_PBResetEp,
	IN_MaskEn 			:= TRUE,
	IO 					:= IO_215DSF,
	HMI 				:= HMI_215DSF
	);

	//LDP UP Limit M6
	_216DSF(
	IN_ConfigPresent 	:= _216DSF.IN_ConfigPresent,
	IN_OnDelay			:= T#1s,
	IN_OffDelay			:= T#1s,
	IN_SwitchDelay		:= T#1s,
	IN_Reset	 		:= VAR_DOS_PBResetEp,
	IN_MaskEn 			:= TRUE,
	IO 					:= IO_216DSF,
	HMI 				:= HMI_216DSF
	);

	//LDP DOWN Limit M6
	_217DSF(
	IN_ConfigPresent 	:= _217DSF.IN_ConfigPresent,
	IN_OnDelay			:= T#1s,
	IN_OffDelay			:= T#1s,
	IN_SwitchDelay		:= T#1s,
	IN_Reset	 		:= VAR_DOS_PBResetEp,
	IN_MaskEn 			:= TRUE,
	IO 					:= IO_217DSF,
	HMI 				:= HMI_217DSF
	);

	_210DSX( //ARM In Cleaning Pos
	IN_ConfigPresent 	:= _210DSX.IN_ConfigPresent,
	IN_Alarm 			:= TRUE,
	IN_AlarmOnReq		:= _210DSX.IN_WaitOff,
	IN_AlarmOffReq 		:= _210DSX.IN_WaitOn,
	IN_OnDelay			:= T#2s,
	IN_OffDelay			:= T#2s,
	IN_SwitchDelay		:= T#100ms,
	IN_WaitOn 			:= DOS.DataOut.CopMode,
	IN_WaitOff 			:= NOT DOS.DataOut.CopMode,
	IN_Reset	 		:= VAR_DOS_PBResetEp,
	IN_MaskEn 			:= TRUE,
	IO 					:= IO_210DSX,
	HMI 				:= HMI_210DSX
	);

	_211DSX( //ARM In Production Pos
	IN_ConfigPresent 	:= _211DSX.IN_ConfigPresent,
	IN_Alarm 			:= TRUE,
	IN_AlarmOnReq		:= _211DSX.IN_WaitOff,
	IN_AlarmOffReq 		:= _211DSX.IN_WaitOn,
	IN_OnDelay			:= T#2s,
	IN_OffDelay			:= T#2s,
	IN_SwitchDelay		:= T#100ms,
	IN_WaitOn 			:= NOT DOS.DataOut.CopMode,
	IN_WaitOff 			:= DOS.DataOut.CopMode,
	IN_Reset	 		:= VAR_DOS_PBResetEp,
	IN_MaskEn 			:= TRUE,
	IO 					:= IO_211DSX,
	HMI 				:= HMI_211DSX
	);

	VAR_DOS_CleanArmProdPos		:= _211DSX.OUT;
	VAR_DOS_CleanArmCopPos		:= _210DSX.OUT;
	VAR_DOS_CleanArmCopPosFault := _210DSX.OUT_Alarm OR _211DSX.OUT_Alarm;
END_ACTION
```

#### DOS_InstrPress.st
```iecst
ACTION DOS_InstrPress:
	_210PTF(
	IN_ConfigPresent 	:= _210PTF.IN_ConfigPresent,
	IN_Alarm 			:= TRUE,
	IN_MaskEn 			:= TRUE,
	IN_Reset 			:= VAR_DOS_PBResetEp,
	IO 					:= IO_210PTF,
	HMI 				:= HMI_210PTF
	);

	//_210PTF ALR
	VAR_DOS_NoBotNoFillPressureLow		:= NOT IO_210PTF.DI_Input; //_210PTF.OUT
	VAR_DOS_NoBotNoFillPressureFault	:= _210PTF.OUT_Alarm;
END_ACTION
```

#### DOS_InstrVolume.st
```iecst
ACTION DOS_InstrVolume:
	//FILIPPO

	_205MEF(
	IN_ConfigPresent	:= _205MEF.IN_ConfigPresent,
	IN_Reset			:= AID.DataOut.Reset,
	IN_ActualSP			:= _205MEF.IN_ActualSP,
	IN_Delta			:= Delta_205MEF,
	IO					:= IO_205MEF,
	HMI					:= HMI_205MEF
	);

	_206MEF(
	IN_ConfigPresent	:= _206MEF.IN_ConfigPresent,
	IN_Reset			:= AID.DataOut.Reset,
	IN_ActualSP			:= _206MEF.IN_ActualSP,
	IN_Delta			:= Delta_206MEF,
	IO					:= IO_206MEF,
	HMI					:= HMI_206MEF
	);

	_212DSF( //MAX VOLUME
		IN_ConfigPresent 	:= _212DSF.IN_ConfigPresent,
		IN_OnDelay			:= T#1s,
		IN_OffDelay			:= T#1s,
		IN_SwitchDelay		:= T#1s,
		IN_Reset	 		:= VAR_DOS_PBResetEp,
		IN_MaskEn 			:= TRUE,
		IO 					:= IO_212DSF,
		HMI 				:= HMI_212DSF
		);

	_213DSF( //MIN VOLUME
		IN_ConfigPresent 	:= _213DSF.IN_ConfigPresent,
		IN_OnDelay			:= T#1s,
		IN_OffDelay			:= T#1s,
		IN_SwitchDelay		:= T#1s,
		IN_Reset	 		:= VAR_DOS_PBResetEp,
		IN_MaskEn 			:= TRUE,
		IO 					:= IO_213DSF,
		HMI 				:= HMI_213DSF
		);

	_212DSF.IN_WaitOn	:= VAR_DOS_LiftMMF205SeqMem.Sensor.SensorMaxVolWaitOn;
	_212DSF.IN_WaitOff	:= VAR_DOS_LiftMMF205SeqMem.Sensor.SensorMaxVolWaitOff;
	_213DSF.IN_WaitOn	:= VAR_DOS_LiftMMF205SeqMem.Sensor.SensorLowPosWaitOn;
	_213DSF.IN_WaitOff	:= VAR_DOS_LiftMMF205SeqMem.Sensor.SensorHighPosWaitOff;

END_ACTION
```

#### DOS_InstrFlow.st
```iecst
ACTION DOS_InstrFlow:

	//FSJ201
	FSJ[201](
	IN_ConfigPresent 	:= FSJ[201].IN_ConfigPresent,
	IN_Alarm 			:= VAR_DOS_SEQ.Device.FSJ201.ALR,
	IN_AlarmOnReq		:= VAR_DOS_SEQ.Device.FSJ201.WAIT_OFF,
	IN_AlarmOffReq 		:= VAR_DOS_SEQ.Device.FSJ201.WAIT_ON,
	IN_SwitchDelay 		:= T#500ms,
	IN_WaitOn 			:= VAR_DOS_SEQ.Device.FSJ201.WAIT_ON,
	IN_WaitOff 			:= VAR_DOS_SEQ.Device.FSJ201.WAIT_OFF,
	IN_Reset	 		:= VAR_DOS_PBResetEp,
	IN_MaskEn 			:= TRUE,
	IO 					:= IO_FSJ[201],
	HMI 				:= HMI_FSJ[201]
	);

	//FSJ202
	FSJ[202](
	IN_ConfigPresent 	:= FSJ[202].IN_ConfigPresent,
	IN_Alarm 			:= VAR_DOS_SEQ.Device.FSJ202.ALR,
	IN_AlarmOnReq		:= VAR_DOS_SEQ.Device.FSJ202.WAIT_OFF,
	IN_AlarmOffReq 		:= VAR_DOS_SEQ.Device.FSJ202.WAIT_ON,
	IN_SwitchDelay 		:= T#500ms,
	IN_WaitOn 			:= VAR_DOS_SEQ.Device.FSJ202.WAIT_ON,
	IN_WaitOff 			:= VAR_DOS_SEQ.Device.FSJ202.WAIT_OFF,
	IN_Reset	 		:= VAR_DOS_PBResetEp,
	IN_MaskEn 			:= TRUE,
	IO 					:= IO_FSJ[202],
	HMI 				:= HMI_FSJ[202]
	);
END_ACTION
```

#### DOS_ManualLifting.st
```iecst
ACTION DOS_ManualLifting:
	ComboBoxString(
	IN_ElementsStructure	:= VAR_LiftPositionType.Elements,
	OUT_ComboString			:= ADR(HMI_DOS_LiftPositionTypeCFG)
	);

	HMI_DOS_LiftPosition.Enable := NOT HMI_DOS_SS2P[SS2P_DOS_SelLiftMan].ON AND SFT.DataOut.MachineEmpty AND VAR_DOS_MotorEnable AND NOT MNM.DataOut.MachineRunning AND NOT (VAR_DOS_LiftMoveStep = DSR_Fault); // AND VAR_DOS_ModeWait;

	VAR_LiftPositionType.Elements[0].Name 		:= '@DOS_Not_Selected';
	VAR_LiftPositionType.Elements[0].Present	:= TRUE;
//	VAR_LiftPositionType.Data[0].PhaseType		:= VAR_DOS_MoveInProductionPosition;

	VAR_LiftPositionType.Elements[1].Name 		:= '@DOS_Production_Position';
	VAR_LiftPositionType.Elements[1].Present	:= TRUE;
//	VAR_LiftPositionType.Data[1].PhaseType		:= VAR_DOS_MoveInProductionPosition;

	VAR_LiftPositionType.Elements[2].Name 		:= '@DOS_COP_Position';
	VAR_LiftPositionType.Elements[2].Present	:= TRUE;
//	VAR_LiftPositionType.Data[2].PhaseType		:= VAR_DOS_MoveInCOPPosition;

	VAR_LiftPositionType.Elements[3].Name 		:= '@DOS_CIP_Position';
	VAR_LiftPositionType.Elements[3].Present	:= TRUE;
//	VAR_LiftPositionType.Data[3].PhaseType		:= VAR_DOS_MoveInCIPPosition;

END_ACTION
```
